(*
Nazwa:			P02_Dispencers
Opis:			Stacja dozownikow
Wersja:			v0.1
Data:			2018-10-10
Autor:			DP
Urzadzenia:		
Konfiguracja:	
Info:

*)
PROGRAM P02_Dispencers
VAR_INPUT
	IbDispencer1DropCatcherBackSensor			AT %I*		:BOOL;					//	Czujnik wycofania tacki kropel dozowników
	IbDispencer2DropCatcherBackSensor 			AT %I*		:BOOL;					//	Czujnik wycofania tacki kropel dozowników
	IbDispencer3DropCatcherBackSensor 			AT %I*		:BOOL;					//	Czujnik wycofania tacki kropel dozowników
	IbDispencer4DropCatcherBackSensor 			AT %I*		:BOOL;					//	Czujnik wycofania tacki kropel dozowników
	IbDispencersCatch1SensorValue 				AT %I*		:DINT;					//	Wejscie czujnika otwarcia siłownika chwytania
	IbDispencersCatch2SensorValue				AT %I*		:DINT;					//	Wejscie czujnika otwarcia siłownika chwytania
	IbDispencersCatch3SensorValue				AT %I*		:DINT;					//	Wejscie czujnika otwarcia siłownika chwytania
	IbDispencersCatch4SensorValue				AT %I*		:DINT;					//	Wejscie czujnika otwarcia siłownika chwytania
	IbDispencersDragLeftLeadBefore1UpSensor		AT %I*		:BOOL;					//	Czujnik
	IbDispencersDragLeftLeadAfter1UpSensor		AT %I*		:BOOL;					//	Czujnik
	IbDispencersDragRightLeadBefore1UpSensor	AT %I*		:BOOL;					//	Czujnik
	IbDispencersDragRightLeadAfter1UpSensor		AT %I*		:BOOL;					//	Czujnik
	IbDispencersDragLeftDragUpSensor 			AT %I*		:BOOL;					// 	Czujnik
	IbDispencersDragLeftDragDownSensor 			AT %I*		:BOOL;					// 	Czujnik
	IbDispencersDragRightDragUpSensor 			AT %I*		:BOOL;					// 	Czujnik
	IbDispencersDragRightDragDownSensor 		AT %I*		:BOOL;					// 	Czujnik
	IbDispencersDragLeftDragHomingSensor 		AT %I*		:BOOL;					//	Czujnik bazowania
	IbDispencersDragRightDragHomingSensor 		AT %I*	 	:BOOL;					//	Czujnik bazowania
	IbDispencerAfterCheckFormSensor				AT %I*		:BOOL; 					//	Czujnik po przecionganiu formatek na ukos
	IbDispencer12NoColisionWhenDosingSensor		AT %I*		:BOOL:=TRUE;			//	Czujnik indukcyjny
	IbDispencer34NoColisionWhenDosingSensor		AT %I*		:BOOL:=TRUE;			//	Czujnik indukcyjny
	//EX
	IbTankLevelHighEX									AT %I*:BOOL;
	IbTankLevelLowEX                                    AT %I*:BOOL;
	IbTankLevelExError									AT %I*:BOOL;
END_VAR
VAR
	
	(*******DOZOWNIK 1*********)
	fbDispencer1										: FB_ServoDispencerServoLifter;			//Blok sterujacy dozownikiem nr1
	eDispencer1State									: E_Station; 							// Stan pracy podajnika platynek			
	eDispencer1RunningState								: E_DispencerState; 
	fbDispencer1State									: FB_State;	
	
	tonDispencer1SuckingValveOpenedSensor				: TON;			//Symulacja czujników 
	tonDispencer1DosingValveOpenedSensor				: TON;			//Symulacja czujników 
	tonDispencer1DosingValveClosedSensor				: TON;			//Symulacja czujników 
	tonDispencer1SuckingValveClosedSensor				: TON;
	
	//WEJŚCIA WYJŚCIA SPRZĘTOWE
	//IbDispencer1SuckingValveOpenedSensor AT%I*:BOOL;	(*dok IO-L*)	//Czujnik otwarcia zaworu ssącego dozownika 1
	QbDispencer1DropCatcherValveActuator				:BOOL;			(*Pneu*)		//Otwarcie tacki
	//IbDispencer1SuckingValveClosedSensor AT%I*:BOOL;	(*dok IO-L*)	//Czujnik zamknięcia zaworu ssąceg odozownika 1
	QbDispencer1SuckingValveActuator					:BOOL;				(*Pneu*)		//sterowanie zaworem ssącego (podłaczenie do wyspypneu)
	QbDispencer1DosingValveActuator						:BOOL;				(*Pneu*)		//sterowanie zaworem dozującym (podłaczenie do wyspypneu)
	
	(*******DOZOWNIK 2*********)
	fbDispencer2										: FB_ServoDispencerServoLifter;				//Blok sterujacy dozownikiem nr 1
	eDispencer2State									: E_Station; 							// Stan pracy podajnika platynek			
	eDispencer2RunningState								: E_DispencerState; 
	fbDispencer2State									: FB_State;	
	
	tonDispencer2SuckingValveOpenedSensor				: TON;			//Symulacja czujników 
	tonDispencer2DosingValveOpenedSensor				: TON;			//Symulacja czujników 
	tonDispencer2DosingValveClosedSensor				: TON;			//Symulacja czujników 
	tonDispencer2SuckingValveClosedSensor				: TON;
	
	//WEJŚCIA WYJŚCIA SPRZĘTOWE
	QbDispencer2DropCatcherValveActuator				:BOOL;			(*Pneu*)			//sterowanie tacką kropel(podłaczenie do wyspy pneu)
	//IbDispencer2SuckingValveOpenedSensor AT%I*:BOOL;	(*dok IO-L*)		//Czujnik otwarcia zaworu ssącego dozownika 1
	//IbDispencer2SuckingValveClosedSensor AT%I*:BOOL;	(*dok IO-L*)		//Czujnik zamknięcia zaworu ssącego dozownika 1
	QbDispencer2SuckingValveActuator					:BOOL;				(*Pneu*)			//sterowanie zaworem ssącego(podłaczeniedowyspypneu)
	QbDispencer2DosingValveActuator						:BOOL;				(*Pneu*)			//sterowanie zaworemd ozującym(podłaczeniedowyspypneu)
	QbDispencerDropCatcherSuck							:BOOL;				(*Pneu*)				//Zasysanie płynu z tacek

	(*******DOZOWNIK 3*********)
	fbDispencer3										: FB_ServoDispencerServoLifter;				//Blok sterujacy dozownikiem nr 1
	eDispencer3State									: E_Station; 							// Stan pracy podajnika platynek			
	eDispencer3RunningState								: E_DispencerState; 
	fbDispencer3State									: FB_State;	
	
	tonDispencer3SuckingValveOpenedSensor				: TON;			//Symulacja czujników 
	tonDispencer3DosingValveOpenedSensor				: TON;			//Symulacja czujników 
	tonDispencer3DosingValveClosedSensor				: TON;			//Symulacja czujników 
	tonDispencer3SuckingValveClosedSensor				: TON;
	
	//WEJŚCIA WYJŚCIA SPRZĘTOWE
	QbDispencer3DropCatcherValveActuator				:BOOL;			(*Pneu*)			//Sterowanie tacką kropel(podłaczenie do wyspy pneu)
	//IbDispencer2SuckingValveOpenedSensor AT%I*:BOOL;	(*dok IO-L*)		//Czujnik otwarcia zaworu ssącego dozownika 1
	//IbDispencer2SuckingValveClosedSensor AT%I*:BOOL;	(*dok IO-L*)		//Czujnik zamknięcia zaworu ssącego dozownika 1
	QbDispencer3SuckingValveActuator					:BOOL;				(*Pneu*)			//sterowanie zaworem ssącego(podłaczeniedowyspypneu)
	QbDispencer3DosingValveActuator						:BOOL;				(*Pneu*)			//sterowanie zaworemd ozującym(podłaczeniedowyspypneu)

	(*******DOZOWNIK 4*********)
	fbDispencer4										: FB_ServoDispencerServoLifter;			// Blok sterujacy dozownikiem nr 1
	eDispencer4State									: E_Station; 							// Stan pracy podajnika platynek			
	eDispencer4RunningState								: E_DispencerState; 
	fbDispencer4State									: FB_State;	
	
	tonDispencer4SuckingValveOpenedSensor				: TON;			//Symulacja czujników 
	tonDispencer4DosingValveOpenedSensor				: TON;			//Symulacja czujników 
	tonDispencer4DosingValveClosedSensor				: TON;			//Symulacja czujników 
	tonDispencer4SuckingValveClosedSensor				: TON;
	
	//WEJŚCIA WYJŚCIA SPRZĘTOWE
	QbDispencer4DropCatcherValveActuator				:BOOL;			(*Pneu*)			//sterowanie tacką kropel(podłaczenie do wyspy pneu)
	//IbDispencer2SuckingValveOpenedSensor AT%I*:BOOL;	(*dok IO-L*)		//Czujnik otwarcia zaworu ssącego dozownika 1
	//IbDispencer2SuckingValveClosedSensor AT%I*:BOOL;	(*dok IO-L*)		//Czujnik zamknięcia zaworu ssącego dozownika 1
	QbDispencer4SuckingValveActuator					:BOOL;				(*Pneu*)			//sterowanie zaworem ssącego(podłaczeniedowyspypneu)
	QbDispencer4DosingValveActuator						:BOOL;				(*Pneu*)			//sterowanie zaworemd ozującym(podłaczeniedowyspypneu)
	
	(*******PODNOSNIK TACKI I CHWYTAKA*********)
	fbDispencersCatch1Station							:FB_CatchStationWithSensor;			// Blok stacji chwytaka dozowników
	fbDispencersCatch2Station							:FB_CatchStationWithSensor;			// Blok stacji chwytaka dozowników
	fbDispencersCatch3Station							:FB_CatchStationWithSensor;			// Blok stacji chwytaka dozowników
	fbDispencersCatch4Station							:FB_CatchStationWithSensor;			// Blok stacji chwytaka dozowników
	eDispencersCatch1State								:E_Station; 				// Stan chwytaka stabilizujšcego pod podajnikiem platynek
	eDispencersCatch2State								:E_Station; 				// Stan chwytaka stabilizujšcego pod podajnikiem platynek
	eDispencersCatch3State								:E_Station; 				// Stan chwytaka stabilizujšcego pod podajnikiem platynek
	eDispencersCatch4State								:E_Station; 				// Stan chwytaka stabilizujšcego pod podajnikiem platynek
	eDispencersCatch1RunningState						:E_CatchStationState; 		// Poprzedni stan chwytaka pod podajnikiem nakrętek
	eDispencersCatch2RunningState						:E_CatchStationState; 		// Poprzedni stan chwytaka pod podajnikiem nakrętek
	eDispencersCatch3RunningState						:E_CatchStationState; 		// Poprzedni stan chwytaka pod podajnikiem nakrętek
	eDispencersCatch4RunningState						:E_CatchStationState; 		// Poprzedni stan chwytaka pod podajnikiem nakrętek
	fbDispencersCatch1State								:FB_State;
	fbDispencersCatch2State								:FB_State;
	fbDispencersCatch3State								:FB_State;
	fbDispencersCatch4State								:FB_State;
	
//WEJSCIA I WYJSCIA SPRZETOWE
	QbDispencersCatch1HeightUpCmd 				AT %Q*	:BOOL; 			(*PLC.A17*)		// Wyjście sterujące podnośnikiem chwytaka i tacki dozownika , Silnik w górę
	QbDispencersCatch1HeightDownCmd 			AT %Q*	:BOOL; 		(*PLC.A17*)		// Wyjście sterujące podnośnikiem chwytaka i tacki dozownika, Silnik w dół
	IbDispencersCatch1HeightEncoderPulses 		AT %I*	:BOOL;	(*PLC.A13*)
	
	IbDispencersCatchHeightEncoderSetCDone		AT %I*: BOOL;
	IudiDispencersCatchHeightEncoderCV          AT %I*: UDINT; 
	QbDispencersCatchHeightEncoderSetC 			AT %Q*: BOOL;		
	QudiDispencersCatchHeightEncoderSetCV       AT %Q*: UDINT; 	
	                                            	
	                                            	
	
	
	QbDispencersCatch1Actuator 							:BOOL;					(*Pneu*)		// Wyjście sterujące chwytakiem pod dozownikami
	QbDispencersCatch2Actuator 							:BOOL;					(*Pneu*)		// Wyjście sterujące chwytakiem pod dozownikami
	QbDispencersCatch3Actuator 							:BOOL;					(*Pneu*)		// Wyjście sterujące chwytakiem pod dozownikami
	QbDispencersCatch4Actuator 							:BOOL;					(*Pneu*)		// Wyjście sterujące chwytakiem pod dozownikami

	QbDispencersCatchMaxPressure						:BOOL;				(*Pneu*)			//sterowanie zaworemd ozującym(podłaczeniedowyspypneu)
	
	(*****************SZLABANY*******************)
	fbDispencerGatesStation								:FB_EntranceGatesServo;			// Blok stacji szlabanów 
		
	(*******PRZECIAGANIE**********)
	eDispencersDragLeftStation							: E_Station;
	eDispencersDragLeftRunningStation					: E_DragStationState;
	fbDispencersDragLeftState							: FB_State;
	eDispencersDragRightStation							: E_Station;
	eDispencersDragRightRunningStation					: E_DragStationState;
	fbDispencersDragRightState							: FB_State;	
	fbDispencersDragLeftStation							: FB_FormsDragStepper;	
	fbDispencersDragRightStation						: FB_FormsDragStepper;
	
	//WEJSCIA I WYJSCIA SPRZETOWE
	
	QbDispencersDragLeftDragActuator                   :BOOL;						// Siłownikiem przeciągania (1 faza)
	
	QbDispencersDragLeftLeadBefore1Actuator          :BOOL;							// Siłownikiem prowadzenia przed 1(1 faza)
	QbDispencersDragLeftLeadAfter1Actuator          :BOOL;							// Siłownikiem prowadzenia przed 1(1 faza)
	
	QbDispencersDragRightDragActuator                  :BOOL;						// Siłownikiem przeciągania (1 faza)
	
	QbDispencersDragRightLeadBefore1Actuator          :BOOL;						// Siłownikiem prowadzenia przed 2(1 faza)	
	QbDispencersDragRightLeadAfter1Actuator          :BOOL;							// Siłownikiem prowadzenia przed 1(1 faza)
		
	(**********ZBIORNIKI**************)
	//Zbiornik
	IbTank1LevelLow 							 AT %I* :BOOL; 				(*PLC.A8*)	// Niski poziom masy w zbiorniku
	IbTank2LevelLow 							 AT %I* :BOOL; 				(*PLC.A8*)	// Niski poziom masy w zbiorniku
	QbTank1LevelSensorCalibration 			     AT %Q* :BOOL;  (*PLC.A20*)	// Kalibracja czujnika poziomu leja nr 1
	QbTank2LevelSensorCalibration 				 AT %Q* :BOOL;  (*PLC.A20*)	// Kalibracja czujnika poziomu leja nr 2
	
	
	QbTank1Pressure								 AT %Q* :BOOL;						(*Pneu*)	// Ciśnienie w zbiorniku nr 1
	bTank1LevelLow                                      :BOOL;									// Sygnały sterujące pompy 1 zależnie od ich odwrócenia
	bTank2LevelLow										:BOOL;									// Sygnały sterujące pompy 2 zależnie od ich odwrócenia
	
	//Pompa podająca
	QbTank1PumpStart 							AT %Q*	:BOOL;		(*PLC.A21*)	//Załączenie pompy masy do zbiornika
	QbTank2PumpStart 							AT %Q*	:BOOL;		(*PLC.A21*)	//Załączenie pompy masy do zbiornika
	QbTank3PumpStart 							AT %Q*	:BOOL;		(*PLC.A21*)	//Załączenie pompy masy do zbiornika
	QbTank4PumpStart 							AT %Q*	:BOOL;		(*PLC.A21*)	//Załączenie pompy masy do zbiornika
	IbTank1PumpFuseOK 							AT %I*  :BOOL; 				//Potwierdzenie z zabezpieczenia pompy 1 - OK
	IbTank2PumpFuseOK 							AT %I*  :BOOL; 				//Potwierdzenie z zabezpieczenia pompy 2 - OK
	IbTank3PumpFuseOK 							AT %I*  :BOOL; 				//Potwierdzenie z zabezpieczenia pompy 2 - OK
	IbTank4PumpFuseOK 							AT %I*  :BOOL; 				//Potwierdzenie z zabezpieczenia pompy 2 - OK
		
	(*GRZAŁKA ZBIORNIKA*)
	fbTankHeating										: FB_TankHeating;	
	eTankHeatingState									: E_Station; 					// Stan pracy grzania
	eTankHeatingRunningState							: E_MassHeatingState; 			// Stan pracy grzania
	fbTankHeatingState									: FB_State;
		
	//WEJŚĆIA I WYJŚĆIA SPRZĘTOWE		
	QbTankHeatingPWMOut							AT %Q* :BOOL; 					// Wyjście sterujące temperaturą grzałki
	AInTankHeatingTempCVSensor 					AT %I* :INT; 			// Wartość aktualnej temperatury grzałki
	IbTankHeatingTempSensorFailure 				AT %I* :BOOL;  		// Informacja o uszkodzeniu czujnika temperatury grzałki	
	
	//Mieszadło zbiornika
	IbFuseTankMixerEngineOK						AT %I* :BOOL;	(*PLC.A7*)	//Bezpiecznik silnika mieszadła OK
	IbFuseTankMixerEngineWorking				AT %I* :BOOL;	{warning 'oprogramowac nowy sygnał mieszadla'}			//Potwierdzenie pracy silnika mieszadła OK	
	QbTank1MixerStart 							AT %Q* :BOOL;			(*PLC.A20*)	//Załączenie mieszadła masy do zbiornika
	
	// Zezwolenie na pracę mieszadła zbiornikowego
	tonTank1LevelSensor									: TON;
	
	tofTank2LevelSensor									: TOF;
	tonTank2LevelSensor									: TON;
	
	tonTank1LevelWarning	   							: TON;
	tonTank2LevelWarning	   							: TON;
	
	tonTank1EmptyAlarm									: TON;
	tonTank2EmptyAlarm									: TON;
	rtDispencer1DoseDone								: R_TRIG;
	rtDispencer2DoseDone								: R_TRIG;
	
	tonTankLevelSensorCalibrationLight					: TON;
	tonTankLevelSensorCalibrationDark					: TON;
	
	(**********OSLONA DOZOWNIKOW*************)	
	
	nCalibrationDialog								 	: INT;

	TimerDispencer1Enable								: TOF;
	TimerDispencer2Enable								: TOF;
	TimerDispencer3Enable								: TOF;
	TimerDispencer4Enable								: TOF;		
	
	(*Wykres dozowania*)
	fbDosingChart1										: FB_WriteDataToArrayString;
	fbDosingChart2										: FB_WriteDataToArrayString;
	fbDosingChart3										: FB_WriteDataToArrayString;
	fbDosingChart4										: FB_WriteDataToArrayString;
	fbDosingStChart1									: FB_WriteDataToArrayOfArrays;
	fbDosingStChart2									: FB_WriteDataToArrayOfArrays;
	fbDosingStChart3									: FB_WriteDataToArrayOfArrays;
	fbDosingStChart4									: FB_WriteDataToArrayOfArrays;
	nChartCycleTime										: INT;
	tDelayDispencerValve								: TIME;

	rtEnable											: R_TRIG;

	fbDropCatcherSuck									: FB_Blink_AS;
	nDose1Counter										: INT;
	nDose2Counter										: INT;
	nDose1CounterWhenLowLevel							: INT;
	nDose2CounterWhenLowLevel							: INT;	
	nDoseCounter1										: INT;
	nDoseCounter2										: INT;	
	// Czujnik poziomu masy przewodząco pojmenościowy LiquiPoint FTW33
	// Zmienne akcji ACT_ConductiveMassSensor
	
	bTank1LevelLowConductiveSensor						: BOOL;
	bTank1SensorDiagnosis								: BOOL;     // Diagnostyka czujnika
	IusiTank1SensorValue0						AT%I*	: USINT;
	IusiTank1SensorValue1						AT%I*	: USINT;
	IusiTank1SensorValue2						AT%I*	: USINT;
	IusiTank1SensorValue3						AT%I*	: USINT;
	IusiTank1SensorDiagnosis					AT%I*	: USINT;
    iTank1Sensor1Value									: INT;	                         
	tonTank1LevelLowConductiveSensor					: TON;
	iTank1Sensor1ValueTemp								: INT;	
	
	bTank2LevelLowConductiveSensor						: BOOL;
	bTank2SensorDiagnosis								: BOOL;     // Diagnostyka czujnika
	IusiTank2SensorValue0						AT%I*	: USINT;
	IusiTank2SensorValue1						AT%I*	: USINT;
	IusiTank2SensorValue2						AT%I*	: USINT;
	IusiTank2SensorValue3						AT%I*	: USINT;
	IusiTank2SensorDiagnosis					AT%I*	: USINT;    
	iTank2Sensor1Value									: INT;		                              
	tonTank2LevelLowConductiveSensor					: TON;	
	iTank2Sensor1ValueTemp								: INT;
	
	//Filtrowanie sygnału
	fbFilterExiTank1Sensor1Value						: FB_FilterEx;
	
	tonMixerNotWorking									: TON;
	
	tonTank1PumpFuseOK									: TON;
	tonTank2PumpFuseOK									: TON;
	
	// Pomocnicze do hamulców
	bDispencer1ManualBrakeOff							: BOOL;
	bDispencer2ManualBrakeOff							: BOOL;	
	bDispencer3ManualBrakeOff							: BOOL;
	bDispencer4ManualBrakeOff							: BOOL;
	
	aDispenser1VirtualLifter							: AXIS_REF;
	aDispenser2VirtualLifter							: AXIS_REF;
	aDispenser3VirtualLifter							: AXIS_REF;
	aDispenser4VirtualLifter							: AXIS_REF;
	
	bDispencer1WithLifter								: BOOL;
	bDispencer2WithLifter								: BOOL;
	bDispencer3WithLifter								: BOOL;
	bDispencer4WithLifter								: BOOL;
	bDispenser1LifterMaster								: BOOL;
	bDispenser2LifterMaster								: BOOL;
	bDispenser3LifterMaster								: BOOL;
	bDispenser4LifterMaster								: BOOL;	
	
	bDispencer12MultiMasterSync							: BOOL;  //Do synchronizacji dozownikow 1-2 miedzy sobą
	bDispencer34MultiMasterSync							: BOOL;	//Do synchornizacji dozownikow 3-4 między sobą
	//bDispencersSyncSim									:BOOL;
	bDispenser1MultiMasterSyncOut						: BOOL;	// Wyjscie synchronizacji dozownika z pozostałymi dozownikami na podnośniku
	bDispenser2MultiMasterSyncOut						: BOOL;	// Wyjscie synchronizacji dozownika z pozostałymi dozownikami na podnośniku
	bDispenser3MultiMasterSyncOut						: BOOL;	// Wyjscie synchronizacji dozownika z pozostałymi dozownikami na podnośniku
	bDispenser4MultiMasterSyncOut						: BOOL;	// Wyjscie synchronizacji dozownika z pozostałymi dozownikami na podnośniku
	
	bDispencer1Manual									: BOOL;
	bDispencer2Manual									: BOOL;
	bDispencer3Manual									: BOOL;
	bDispencer4Manual									: BOOL;
	
	bDispencer1DropCatcherValveActuator					: BOOL;
	bDispencer2DropCatcherValveActuator					: BOOL;
	bDispencer3DropCatcherValveActuator					: BOOL;
	bDispencer4DropCatcherValveActuator					: BOOL;
	
	ftChangeover										: F_TRIG;
	
	//Mikołaj
	
	rtbDispencer12EnableShow							: R_TRIG;
	ftbDispencer12EnableShow							: F_TRIG;
	rtbDispencer34EnableShow							: R_TRIG;
	ftbDispencer34EnableShow							: F_TRIG;
	
	fbDispencersCleaningPID								: FB_PIDBasic;
	tonbDispencer12Cleaning								: TON;
	tonbDispencer34Cleaning								: TON;	
	fbDispencersCIP										: FB_InputFilter;

	ftCIP												: F_TRIG;
	tonbCIP												: TON;
	ftbCIP												: F_TRIG;
	rtbCIP												: R_TRIG;
	
	tonResetOpenCalibration								: TON;
	tonResetCloseCalibration							: TON;
	
	tofDispencersDragLeftStationEnable					: TOF;
	tofDispencersDragRightStationEnable					: TOF;	
	
	
	fbFormsDragingStepperState: INT;
	eState: INT;

	tofTank1LevelSensor: TOF;
//dodane filtry 	
	fbIbDispencer1DropCatcherBackSensor	:FB_InputFilter;
	fbIbDispencer2DropCatcherBackSensor	:FB_InputFilter;
	fbIbDispencer3DropCatcherBackSensor	:FB_InputFilter;
	fbIbDispencer4DropCatcherBackSensor	:FB_InputFilter;
		
	arTemp:AXIS_REF;

	(*Tryb serwisowy dozownikow*)
	ftbDispencersPullingSlow: F_TRIG;
	ftbDispencersPullingFast: F_TRIG;
	ftbDispencersPullingSlowContinous: F_TRIG;
	ftbDispencersPullingFastContinous: F_TRIG;	
	ftbDispencersLifterUp: F_TRIG;
	ftbDispencersLifterDown: F_TRIG;
	tonbDispencersPullingContinous: TON;

	rtDispencer1Sync												: R_TRIG;
	rtDispencer2Sync												: R_TRIG;
	rtDispencer3Sync												: R_TRIG;
	rtDispencer4Sync												: R_TRIG;
	fbDispencer1Sync												: FB_InputFilter_v2;	
	fbDispencer2Sync												: FB_InputFilter_v2;	
	fbDispencer3Sync												: FB_InputFilter_v2;	
	fbDispencer4Sync												: FB_InputFilter_v2;	
	tofDispencersSync												: TOF;
	rtManualMode													: R_TRIG;
	ftManualMode													: F_TRIG;
	rtbDispencer1Sync												: R_TRIG;	
	rtbDispencer2Sync												: R_TRIG;		
	rtbDispencer3Sync												: R_TRIG;	
	rtbDispencer4Sync												: R_TRIG;	
	rtbDispencer12Sync												: R_TRIG;
	rtbDispencer34Sync												: R_TRIG;
	rtbDispencer1234Sync											: R_TRIG;	
	rtHeightSetDispencer12											: R_TRIG;
	rtHeightSetDispencer34											: R_TRIG;

	bDispencer1SyncTemp												: BOOL;
	bDispencer2SyncTemp												: BOOL;
	bDispencer3SyncTemp												: BOOL;
	bDispencer4SyncTemp												: BOOL;
	
	(*Reset warningów*)
	tonDispencersWarningReset : TON;
	
	(*Podtrzymanie receptur*)
	bFormsDragingLeftEnableDelay: BOOL;
	bFormsDragingRightEnableDelay: BOOL;
	bDispencer1EnableDelay: BOOL;
	bDispencer2EnableDelay: BOOL;
	bDispencer3EnableDelay: BOOL;
	bDispencer4EnableDelay: BOOL;
	
	(*inne*)
	btemp					:BOOL;
	
	(*Ex*)
	tonLowLevelExSensor		:TON;
	tonErrorExSensorDelay	:TON;
	bTank1LevelExSensor: BOOL;	

	//Zmienne od EVENTLOGGER
	bAlarmInit 						: BOOL := TRUE; 
	nAlarmNumerator					: INT;
	arfbAlarm						: ARRAY[0..19] OF  FB_TcAlarm;		//Tablica bloczków błędów
	fbSourceInfo 					: FB_TcSourceInfo;
	iSourceInfo						: I_TcSourceInfo;
	sAlarmTest						: STRING;
	//Koniec zmiennych od EVENTLOGGER
END_VAR

(* Temp zbiornika*)
VIS.lrTankHeatingTempCV := AInTankHeatingTempCVSensor/10.0;
(* Koniec Temp zbiornika*)

fbIbDispencer1DropCatcherBackSensor(bIN:=IbDispencer1DropCatcherBackSensor AND IbDispencer2DropCatcherBackSensor ,tFilterTimeOn:=T#20MS,tFilterTimeOff:=T#20MS,bOUT=>);
fbIbDispencer2DropCatcherBackSensor(bIN:=IbDispencer2DropCatcherBackSensor AND IbDispencer1DropCatcherBackSensor,tFilterTimeOn:=T#20MS,tFilterTimeOff:=T#20MS,bOUT=>);
fbIbDispencer3DropCatcherBackSensor(bIN:=IbDispencer3DropCatcherBackSensor AND IbDispencer4DropCatcherBackSensor,tFilterTimeOn:=T#20MS,tFilterTimeOff:=T#20MS,bOUT=>);
fbIbDispencer4DropCatcherBackSensor(bIN:=IbDispencer4DropCatcherBackSensor AND IbDispencer3DropCatcherBackSensor,tFilterTimeOn:=T#20MS,tFilterTimeOff:=T#20MS,bOUT=>);
	


(***Skalownaie wartości zadanej na 1-100%************)
(*
:=DINT_TO_USINT(
	F_Scaling(
	rValue:= LREAL_TO_DINT(lrFormsDragingLeftVelocity), 
	rXmin:= 1, 
	rXmax:= 1000, 
	rYmin:= 1, 
	rYmax:= 10)
	)
;*)


fbDispencersCatch1Station.lrSensorTolerance:= fbDispencersCatch2Station.lrSensorTolerance:= 
fbDispencersCatch3Station.lrSensorTolerance:= fbDispencersCatch4Station.lrSensorTolerance:= 
	F_Scaling(
	rValue:= LREAL_TO_DINT(lrDispencersCatchTolerance*10), 
	rXmin:= 1, 
	rXmax:= 100, 
	rYmin:= 100, 
	rYmax:= 10000)
;

IF lrDispencersCatchTolerance = 100 THEN
	fbDispencersCatch1Station.lrSensorTolerance	:= fbDispencersCatch2Station.lrSensorTolerance	:= 100000;	
	fbDispencersCatch3Station.lrSensorTolerance	:= fbDispencersCatch4Station.lrSensorTolerance	:= 100000;	
END_IF
(****Koniec skalownaie wartości zadanej na 1-100%****)

//Grzanie zbiornika
IF NOT VIS.bLidFeederEnableShow THEN
	//GVL.bDispencersCatchEnable																		:= NOT VIS.bSimulation ;
END_IF
(**SYMULACJA CZUJNIKÓW IGLIC**)
tDelayDispencerValve																			:= T#50MS;

tonDispencer1SuckingValveClosedSensor(IN:=NOT QbDispencer1SuckingValveActuator, PT:=tDelayDispencerValve);
tonDispencer1SuckingValveOpenedSensor(IN:=QbDispencer1SuckingValveActuator,PT:=tDelayDispencerValve);
tonDispencer1DosingValveOpenedSensor(IN:=QbDispencer1DosingValveActuator ,PT:=tDelayDispencerValve);
tonDispencer1DosingValveClosedSensor(IN:=NOT QbDispencer1DosingValveActuator ,PT:=tDelayDispencerValve);

tonDispencer2SuckingValveClosedSensor(IN:=NOT QbDispencer2SuckingValveActuator, PT:=tDelayDispencerValve);
tonDispencer2SuckingValveOpenedSensor(IN:=QbDispencer2SuckingValveActuator,PT:=tDelayDispencerValve);
tonDispencer2DosingValveOpenedSensor(IN:=QbDispencer2DosingValveActuator ,PT:=tDelayDispencerValve);
tonDispencer2DosingValveClosedSensor(IN:=NOT QbDispencer2DosingValveActuator ,PT:=tDelayDispencerValve);

tonDispencer3SuckingValveClosedSensor(IN:=NOT QbDispencer3SuckingValveActuator, PT:=tDelayDispencerValve);
tonDispencer3SuckingValveOpenedSensor(IN:=QbDispencer3SuckingValveActuator,PT:=tDelayDispencerValve);
tonDispencer3DosingValveOpenedSensor(IN:=QbDispencer3DosingValveActuator ,PT:=tDelayDispencerValve);
tonDispencer3DosingValveClosedSensor(IN:=NOT QbDispencer3DosingValveActuator ,PT:=tDelayDispencerValve);

tonDispencer4SuckingValveClosedSensor(IN:=NOT QbDispencer4SuckingValveActuator, PT:=tDelayDispencerValve);
tonDispencer4SuckingValveOpenedSensor(IN:=QbDispencer4SuckingValveActuator,PT:=tDelayDispencerValve);
tonDispencer4DosingValveOpenedSensor(IN:=QbDispencer4DosingValveActuator ,PT:=tDelayDispencerValve);
tonDispencer4DosingValveClosedSensor(IN:=NOT QbDispencer4DosingValveActuator ,PT:=tDelayDispencerValve);
(**Koniec SYMULACJA CZUJNIKÓW IGLIC*)

aLimits();
aAntyColision();
aDispencersEnable();
aCleaning();
aDispencersLiftersBefore(); //musi być odpowednia kolejność 
aDispencersManualMode();
aDispencer1();
aDispencer2();
aDispencer3();
aDispencer4();
aDispencersLiftersAfter();
aDispencerCatch1();
aDispencerCatch2();
aDispencerCatch3();
aDispencerCatch4();
aDispencerCatchPressure();
aDispencersCatchWarnings();
aDropCatcher();
aDispencerDragStation();
aDispencersDragStationLeadActuators();
aTanks();
aTanksRainbowMode();
aTankWarning();
aTankHeating();
aTDRMassSensor();
aExSensor();
aLevelSensorCalibration();
aDosingChartHMI(); //Przygotowanie danych do wykresu

(* BAZOWANIE - ZMIAN*)
rtEnable		(CLK:=fbDispencer1.bEnable OR fbDispencer2.bEnable OR fbDispencer3.bEnable OR fbDispencer4.bEnable,				Q=>);
ftChangeover	(CLK:=fbDispencer1.bChangeover OR fbDispencer2.bChangeover OR fbDispencer2.bChangeover OR fbDispencer2.bChangeover, Q=>);
ftCIP			(CLK:=bCIP, 																									Q=>);

IF ( rtEnable.Q  OR ftChangeover.Q OR ftCIP.Q) AND (P00_PackML.fbPMLAuto.ePMLState = E_PMLState.ePMLState_IDLE OR P00_PackML.fbPMLAuto.ePMLState = E_PMLState.ePMLState_EXECUTE)  THEN
	VIS.bDispencer12LifterHeightSet:=TRUE;
	VIS.bDispencer34LifterHeightSet:=TRUE;	
	VIS.bDispencersCatchHeightSet:=TRUE;
	
ELSIF ( fbDispencer1.eState=E_Station.eHomingDone AND 
		fbDispencer2.eState=E_Station.eHomingDone AND 
		fbDispencer3.eState=E_Station.eHomingDone AND 
		fbDispencer4.eState=E_Station.eHomingDone) OR 
		VIS.bErrorOccure THEN
	VIS.bDispencer12LifterHeightSet:=FALSE;
	VIS.bDispencer34LifterHeightSet:=FALSE;
ELSIF fbDispencersCatch1Station.eState=E_Station.eHomingDone OR VIS.bErrorOccure THEN
	VIS.bDispencersCatchHeightSet:=FALSE;
ELSIF fbDispencer1.eState=E_Station.eHomingDone OR VIS.bErrorOccure THEN
	VIS.bDispencer12LifterHeightSet:=FALSE;
ELSIF fbDispencer2.eState=E_Station.eHomingDone OR VIS.bErrorOccure THEN
	VIS.bDispencer12LifterHeightSet:=FALSE;
ELSIF fbDispencer3.eState=E_Station.eHomingDone OR VIS.bErrorOccure THEN
	VIS.bDispencer34LifterHeightSet:=FALSE;
ELSIF fbDispencer4.eState=E_Station.eHomingDone OR VIS.bErrorOccure THEN
	VIS.bDispencer34LifterHeightSet:=FALSE;

END_IF


(********* GENEROWANIE STANU STACJI DO WIZKI**********)
fbDispencersDragLeftState(
	eState:=eDispencersDragLeftStation, 
	bRun:=VIS.bFormsDragingLeftRun,
	eFormsDragingRunningState:=eDispencersDragLeftRunningStation , 
	sStateDesc=> VIS.sFormsDragingLeftState,
	iState=>VIS.iFormsDragingLeftState);
fbDispencersDragRightState(
	eState:=eDispencersDragRightStation, 
	bRun:=VIS.bFormsDragingRightRun,
	eFormsDragingRunningState:=eDispencersDragRightRunningStation , 
	sStateDesc=> VIS.sFormsDragingRightState,
	iState=>VIS.iFormsDragingRightState);	
fbDispencer1State(
	eState:=eDispencer1State , 
	bRun:=VIS.bDispencer1Dose,
	eDispencerRunningState:=eDispencer1RunningState , 
	sStateDesc=> VIS.sDispencer1State,
	iState=>VIS.iDispencer1State);
fbDispencer2State(
	eState:=eDispencer2State , 
	bRun:=VIS.bDispencer2Dose,
	eDispencerRunningState:=eDispencer2RunningState , 
	sStateDesc=> VIS.sDispencer2State,
	iState=>VIS.iDispencer2State);
fbDispencer3State(
	eState:=eDispencer3State , 
	bRun:=VIS.bDispencer3Dose,
	eDispencerRunningState:=eDispencer3RunningState , 
	sStateDesc=> VIS.sDispencer3State,
	iState=>VIS.iDispencer3State);
fbDispencer4State(
	eState:=eDispencer4State , 
	bRun:=VIS.bDispencer4Dose,
	eDispencerRunningState:=eDispencer4RunningState , 
	sStateDesc=> VIS.sDispencer4State,
	iState=>VIS.iDispencer4State);
fbDispencersCatch1State(
	eState:=eDispencersCatch1State	 , 
	bRun:=VIS.bDispencers1Catch,	
	eCatchRunningState:=eDispencersCatch1RunningState , 
	sStateDesc=> VIS.sDispencersCatch1State,
	iState=>VIS.iDispencersCatch1State	);		
fbDispencersCatch2State(
	eState:=eDispencersCatch2State	 , 
	bRun:=VIS.bDispencers2Catch,	
	eCatchRunningState:=eDispencersCatch2RunningState , 
	sStateDesc=> VIS.sDispencersCatch2State,
	iState=>VIS.iDispencersCatch2State	);	
fbDispencersCatch3State(
	eState:=eDispencersCatch3State	 , 
	bRun:=VIS.bDispencers3Catch,	
	eCatchRunningState:=eDispencersCatch3RunningState , 
	sStateDesc=> VIS.sDispencersCatch3State,
	iState=>VIS.iDispencersCatch3State	);	
fbDispencersCatch4State(
	eState:=eDispencersCatch4State	 , 
	bRun:=VIS.bDispencers4Catch,	
	eCatchRunningState:=eDispencersCatch4RunningState , 
	sStateDesc=> VIS.sDispencersCatch4State,
	iState=>VIS.iDispencersCatch4State	);		
fbTankHeatingState(
	eState:=eTankHeatingState, 
	bRun:=bTankHeatingEnable,
	eMassHeatingRunningState:=eTankHeatingRunningState , 
	);
(***** KONIEC GENEROWANIE STANU STACJI DO WIZKI*******)


(**Przypisanie maksymalnej prędkość podnośników dozowników do ekranu ustawiania wykresu dozowania*)
VIS.iHMIDispencersLifterMaxSpeed := 313;
(**Koniec Przypisanie maksymalnej prędkość podnośników dozowników do ekranu ustawiania wykresu dozowania*)


(******* Wypracowanie sygnałów dla HMI *******)
VIS.lrDispencer1ActPos := aDispencer1AxisRef.NcToPlc.ActPos;
VIS.lrDispencer2ActPos := aDispencer2AxisRef.NcToPlc.ActPos;
VIS.lrDispencer3ActPos := aDispencer3AxisRef.NcToPlc.ActPos;
VIS.lrDispencer4ActPos := aDispencer4AxisRef.NcToPlc.ActPos;

(*******Jezeli dwufazowe to przepisuj sygnały**************)


IF NOT VIS.bDosingTwoPhasesShow THEN
	VIS.lrDispencer2DoseVolumeShow:=VIS.lrDispencer1DoseVolumeShow;
	VIS.lrDispencer2Phase1VolumeShow:=VIS.lrDispencer1Phase1VolumeShow;
	VIS.lrDispencer2Phase2VolumeShow:=VIS.lrDispencer1Phase2VolumeShow;
	VIS.lrDispencer2Phase1VelocityShow:=VIS.lrDispencer1Phase1VelocityShow;
	VIS.lrDispencer2Phase2VelocityShow:=VIS.lrDispencer1Phase2VelocityShow;
	VIS.lrDispencer2Phase3VelocityShow:=VIS.lrDispencer1Phase3VelocityShow;
	VIS.lrDispencer2SuckVelocityShow:=VIS.lrDispencer1SuckVelocityShow;
	VIS.lrDispencer2Phase1AccelerationShow:=VIS.lrDispencer1Phase1AccelerationShow;
	VIS.lrDispencer2Phase2AccelerationShow:=VIS.lrDispencer1Phase2AccelerationShow;
	VIS.lrDispencer2Phase3AccelerationShow:=VIS.lrDispencer1Phase3AccelerationShow;
	VIS.lrDispencer2SuckAccelerationShow:=VIS.lrDispencer1SuckAccelerationShow;
	VIS.lrDispencer2Phase1DecelerationShow:=VIS.lrDispencer1Phase1DecelerationShow;
	VIS.lrDispencer2Phase2DecelerationShow:=VIS.lrDispencer1Phase2DecelerationShow;
	VIS.lrDispencer2Phase3DecelerationShow:=VIS.lrDispencer1Phase3DecelerationShow;
	VIS.udiDispencer2DosingDoneDelayTimeShow:=VIS.udiDispencer1DosingDoneDelayTimeShow;
	VIS.lrDispencer2SuckValveOpenVolumeShow:=VIS.lrDispencer1SuckValveOpenVolumeShow;
	VIS.lrDispencer2SuckValveOpenTimeDelayShow:=VIS.lrDispencer1SuckValveOpenTimeDelayShow;
	VIS.lrDispencer2SuckValveCloseVolumeShow:=VIS.lrDispencer1SuckValveCloseVolumeShow;
	VIS.lrDispencer2SuckValveCloseTimeDelayShow:=VIS.lrDispencer1SuckValveCloseTimeDelayShow;
	VIS.lrDispencer2DoseValveOpenVolumeShow:=VIS.lrDispencer1DoseValveOpenVolumeShow;
	VIS.lrDispencer2DoseValveOpenTimeAccShow:=VIS.lrDispencer1DoseValveOpenTimeAccShow;
	VIS.lrDispencer2DoseValveCloseVolumeShow:=VIS.lrDispencer1DoseValveCloseVolumeShow;
	VIS.lrDispencer2DoseValveCloseTimeDecShow:=VIS.lrDispencer1DoseValveCloseTimeDecShow;
	VIS.lrDispencer2DoseSuckingVolumeShow:=VIS.lrDispencer1DoseSuckingVolumeShow;
	VIS.lrDispencer2DoseSuckingTimeDelayShow:=VIS.lrDispencer1DoseSuckingTimeDelayShow;
	VIS.bDispencer2DoseSuckingShow:=VIS.bDispencer1DoseSuckingShow;
	VIS.bDispencer2LiftSynchroPh1Show:=VIS.bDispencer1LiftSynchroPh1Show;
	VIS.bDispencer2LiftSynchroPh2Show:=VIS.bDispencer1LiftSynchroPh2Show;
	VIS.bDispencer2LiftSynchroPh3Show:=VIS.bDispencer1LiftSynchroPh3Show;
	VIS.lrDispencer2LifterStartDosePositionShow:=VIS.lrDispencer1LifterStartDosePositionShow;
	VIS.lrDispencer2LifterStopDosePositionShow:=VIS.lrDispencer1LifterStopDosePositionShow;
	VIS.lrDispencer2LifterVelocityShow:=VIS.lrDispencer1LifterVelocityShow;
	VIS.lrDispencer2LifterAccelerationShow:=VIS.lrDispencer1LifterAccelerationShow;
	VIS.lrDispencer2LifterDecelerationShow:=VIS.lrDispencer1LifterDecelerationShow;
	
//dodane po testach 	
	VIS.lrFormsDragingRightAccelerationShow:=VIS.lrFormsDragingLeftAccelerationShow;
	VIS.lrFormsDragingRightDecelerationShow:=VIS.lrFormsDragingLeftDecelerationShow;
	VIS.lrFormsDragingRightVelocityShow:=VIS.lrFormsDragingLeftVelocityShow;
	
END_IF

IF bCycleReseting THEN
	;
END_IF


(*Opoznienie wyłączanie enabla dozownikow*)
(*Nie zdarzy wyjśc z Disabled podczas zmiany recepptury*)
TimerDispencer1Enable(IN:=bDispencer1Enable OR bDispencer1EnableDelay, PT:=T#5S);
TimerDispencer2Enable(IN:=bDispencer2Enable OR bDispencer2EnableDelay, PT:=T#5S);
TimerDispencer3Enable(IN:=bDispencer3Enable OR bDispencer3EnableDelay, PT:=T#5S);
TimerDispencer4Enable(IN:=bDispencer4Enable OR bDispencer4EnableDelay, PT:=T#5S);
// Dodatkowe podtrzymanie przy zmianie receptury
IF  P00_PackML.fbbRecipeLoading.bOut AND GVL.bDispencer1Enable	THEN	bDispencer1EnableDelay	:= 	TRUE;	END_IF
IF  P00_PackML.fbbRecipeLoading.bOut AND GVL.bDispencer2Enable	THEN	bDispencer2EnableDelay	:= 	TRUE;	END_IF
IF  P00_PackML.fbbRecipeLoading.bOut AND GVL.bDispencer3Enable	THEN	bDispencer3EnableDelay	:= 	TRUE;	END_IF
IF  P00_PackML.fbbRecipeLoading.bOut AND GVL.bDispencer4Enable	THEN	bDispencer4EnableDelay	:= 	TRUE;	END_IF
IF NOT P00_PackML.fbbRecipeLoading.bOut THEN
	bDispencer1EnableDelay	:= FALSE;
	bDispencer2EnableDelay	:= FALSE;
	bDispencer3EnableDelay	:= FALSE;	
	bDispencer4EnableDelay	:= FALSE;	
END_IF
// Koniec podtrzymanie przy zmianie receptury






(********KASOWANIE ROZKAZÓW CYKLI*********)
IF fbDispencer1.bCycleDone AND bManualMode THEN
	VIS.bDispencer1Dose := FALSE;
END_IF
IF fbDispencer2.bCycleDone AND bManualMode THEN
	VIS.bDispencer2Dose := FALSE;
END_IF
IF fbDispencer3.bCycleDone AND bManualMode THEN
	VIS.bDispencer3Dose := FALSE;
END_IF
IF fbDispencer4.bCycleDone AND bManualMode THEN
	VIS.bDispencer4Dose := FALSE;
END_IF
 
(*****KONIEC KASOWANIA ROZKAZÓW CYKLI*****)
tonResetCloseCalibration(IN:= VIS.bDispencersCatchCloseCalibration, PT:= T#3S);
tonResetOpenCalibration	(IN:= VIS.bDispencersCatchOpenCalibration, PT:= T#3S);
IF tonResetOpenCalibration.Q THEN
	VIS.bDispencersCatchOpenCalibration	:= FALSE;
END_IF
IF tonResetCloseCalibration.Q THEN
	VIS.bDispencersCatchCloseCalibration := FALSE;
END_IF


tofDispencersDragLeftStationEnable	(IN:= GVL.bFormsDragingLeftEnable OR bFormsDragingLeftEnableDelay, 		PT:= T#10S);
tofDispencersDragRightStationEnable	(IN:= GVL.bFormsDragingRightEnable OR bFormsDragingRightEnableDelay,	PT:= T#10S);
// Dodatkowe podtrzymanie przy zmianie receptury
IF  P00_PackML.fbbRecipeLoading.bOut AND GVL.bFormsDragingLeftEnable	THEN	bFormsDragingLeftEnableDelay	:= 	TRUE;	END_IF
IF  P00_PackML.fbbRecipeLoading.bOut AND GVL.bFormsDragingRightEnable	THEN	bFormsDragingRightEnableDelay	:= 	TRUE;	END_IF
IF NOT P00_PackML.fbbRecipeLoading.bOut THEN
	bFormsDragingLeftEnableDelay	:= FALSE;
	bFormsDragingRightEnableDelay	:= FALSE;
END_IF
// Koniec podtrzymanie przy zmianie receptury


IF fbDispencersDragLeftStation.bCycleDone AND bManualMode THEN
	VIS.bFormsDragingLeftRun 									:= FALSE;
	GVL.bFormsDragingLeftPrepareRun								:= FALSE;
END_IF
IF fbDispencersDragRightStation.bCycleDone AND bManualMode THEN
	VIS.bFormsDragingRightRun 									:= FALSE;
	GVL.bFormsDragingRightPrepareRun							:= FALSE;
END_IF

ACTION aAntyColision:

//Pozycja MIN dla dozowników
IF VIS.lrDispencersCatchHeightCV-200 > 40 THEN
	fbDispencer1.lrMinPosition :=	VIS.lrDispencersCatchHeightCV-200;
	fbDispencer2.lrMinPosition :=	VIS.lrDispencersCatchHeightCV-200;
	fbDispencer3.lrMinPosition :=	VIS.lrDispencersCatchHeightCV-200;
	fbDispencer4.lrMinPosition :=	VIS.lrDispencersCatchHeightCV-200;
ELSE
	fbDispencer1.lrMinPosition :=	40;
END_IF

//Pozycja MAX dla chwytaka
IF VIS.lrDispencer12LifterActPos < VIS.lrDispencer34LifterActPos THEN
	fbDispencersCatch1Station.lrMaxHeight := VIS.lrDispencer12LifterActPos + 200;
ELSE
	fbDispencersCatch1Station.lrMaxHeight := VIS.lrDispencer34LifterActPos + 200;
END_IF
END_ACTION

ACTION aCleaning:
(*** MYCIE DOZOWNIKÓW CIP 12***)
(* Doza naprzemienna i pompowanie zbiornika*)

//Zmienne
VIS.bDispencersCIP;		//Włączony CIP z wizu
bCIP;					//Przefiltrowany sygnał CIP
VIS.iDispencersCIP;		//Informacja o ruchu wylewek
VIS.bDispencer12Cleaning;
VIS.bDispencer34Cleaning;
eDispencer1RunningState;		aDispencer1AxisRef.NcToPlc.ActPos;
eDispencer2RunningState;		aDispencer2AxisRef.NcToPlc.ActPos;
VIS.bDispencer12Cleaning;		bDispencer1Cleaning;bDispencer2Cleaning;
VIS.lrDispencersManualOverride;


//Filtrowanie sygnału, przeciw lagom z wizualizacji lub ciągłym klikaniem
fbDispencersCIP(bIn:=VIS.bDispencersCIP,tFilterTimeOn:=T#0MS,tFilterTimeOff:=T#3S,bOUT=>bCIP);

tonbCIP	(IN:=bCIP, PT:=T#7S);
ftbCIP	(CLK:=bCIP,	Q=>);
rtbCIP	(CLK:=bCIP,	Q=>);

IF rtbCIP.Q THEN
	VIS.bTank1SupplyPumpEnableShow:=FALSE;
	VIS.bTank2SupplyPumpEnableShow:=FALSE;
END_IF

//Przejazd chwytaków i dozowników
IF bCIP THEN
	VIS.bDispencer12ManualLifterDown	:= VIS.lrDispencer12LifterActPos	>	40;
	VIS.bDispencer34ManualLifterDown	:= VIS.lrDispencer34LifterActPos	>	40;
	VIS.iDispencersCIP := 0;
	IF tonbCIP.Q THEN // Ustawianie informacji o stacji z opóźnieniem
		IF P02_Dispencers.fbDispencersCatch1Station.eState = E_Station.ePreparingToDisable OR P02_Dispencers.fbDispencersCatch1Station.eState = E_Station.eHoming
		OR VIS.bDispencer12ManualLifterDown OR VIS.bDispencer34ManualLifterDown
		THEN
			VIS.iDispencersCIP 			:=	0;
		ELSIF P02_Dispencers.fbDispencersCatch1Station.eState = E_Station.eDisabled THEN
			VIS.iDispencersCIP 			:=	-1;
		END_IF 
	END_IF
END_IF

//Kasowanie rozkazów na wszelki wypadek
IF ftbCIP.Q THEN
	VIS.bDispencer12ManualLifterDown 		:= FALSE;
	VIS.bDispencer34ManualLifterDown 		:= FALSE;
	VIS.bDispencer1ManualSuckValve			:= FALSE;
	VIS.bDispencer1ManualDoseValve			:= FALSE;
	VIS.bDispencer2ManualSuckValve			:= FALSE;
	VIS.bDispencer2ManualDoseValve			:= FALSE;
	VIS.bDispencer3ManualSuckValve			:= FALSE;
	VIS.bDispencer3ManualDoseValve			:= FALSE;
	VIS.bDispencer4ManualSuckValve			:= FALSE;
	VIS.bDispencer4ManualDoseValve			:= FALSE;
	VIS.iDispencersCIP := 0;
END_IF


//PID regulacji poziomu
fbDispencersCleaningPID(
	bEnable:= VIS.bDispencer12Cleaning OR VIS.bDispencer34Cleaning , 
	bInvertDirection:=TRUE , 
	lrSetpointValue:= 20, 
	lrActualValue:= iTank1Sensor1Value, 
	bReset:= , 
	lrYMin:= 50, 
	lrYMax:= 100, 
	lrKp:= 0.0001, 
	tTn:= T#10S, 
	tTv:= , 
	tTd:=T#0S , 
	lrTaskCycleTime:=10.0 , 
	lrCycleTime:= 1000, 
	lrY=> , 
	bError=> );
 
//Wyłączenie mycia CIP po czasie	
tonbDispencer12Cleaning(IN:=VIS.bDispencer12Cleaning, PT:=T#360S);
IF tonbDispencer12Cleaning.Q THEN
	VIS.bDispencer12Cleaning := FALSE;
END_IF
tonbDispencer34Cleaning(IN:=VIS.bDispencer34Cleaning, PT:=T#360S);
IF tonbDispencer34Cleaning.Q THEN
	VIS.bDispencer34Cleaning := FALSE;
END_IF


IF VIS.bTank1ManualSupplyPump AND VIS.bTank1LevelSensorHigh AND VIS.iTank1LevelSensorValue>110 THEN
	VIS.bTank1ManualSupplyPump := FALSE;
END_IF

//DOZOWNIKI 1 i 2 | Procedura mycia CIP
IF VIS.bDispencer12Cleaning THEN
	//Ustawienie njaniższego poziomu w zbiorniku
	VIS.uTank1LevelSetpointShow;VIS.bTank1LevelSensorLow;VIS.bTank1LevelSensorHigh; //Ustawianie w aTanks
	//Włączenie pompy
	VIS.bTank1SupplyPumpEnableShow;VIS.bTank1ManualSupplyPump;
	//Ustawienie override od PIDa
	//VIS.lrDispencerManualOverride	:= fbDispencersCleaningPID.lrY; 
	//Dozownaie naprzemienne
	IF eDispencer1RunningState = E_DispencerState.eCleaningReady  THEN
	 	bDispencer1Cleaning 		:=	TRUE;
	END_IF	
	IF eDispencer2RunningState = E_DispencerState.eCleaningReady  AND (eDispencer1RunningState = E_DispencerState.eCleaning AND aDispencer1AxisRef.NcToPlc.ActPos < 100) THEN
		bDispencer2Cleaning 		:=	TRUE;
	END_IF
	IF eDispencer1RunningState = E_DispencerState.eCleaningDone  THEN
	 	bDispencer1Cleaning 		:=	FALSE;
	END_IF
	IF eDispencer2RunningState = E_DispencerState.eCleaningDone  THEN
	 	bDispencer2Cleaning 		:=	FALSE;
	END_IF		
ELSE //Czyszczenie 
	 bDispencer1Cleaning			:= bDispencer2Cleaning	:=	FALSE;
END_IF

//DOZOWNIKI 3 i 4 | Procedura mycia CIP
IF VIS.bDispencer34Cleaning THEN
	//Ustawienie njaniższego poziomu w zbiorniku
	VIS.uTank1LevelSetpointShow;VIS.bTank1LevelSensorLow;VIS.bTank1LevelSensorHigh; //Ustawianie w aTanks
	//Ustawienie override od PIDa
	//VIS.lrDispencerManualOverride	:= fbDispencersCleaningPID.lrY; 
	//Dozownaie naprzemienne
	IF eDispencer3RunningState = E_DispencerState.eCleaningReady  THEN
	 	bDispencer3Cleaning 		:=	TRUE;
	END_IF	
	IF eDispencer4RunningState = E_DispencerState.eCleaningReady  AND (eDispencer3RunningState = E_DispencerState.eCleaning AND aDispencer3AxisRef.NcToPlc.ActPos < 100) THEN
		bDispencer4Cleaning 		:=	TRUE;
	END_IF
	IF eDispencer3RunningState = E_DispencerState.eCleaningDone  THEN
	 	bDispencer3Cleaning 		:=	FALSE;
	END_IF
	IF eDispencer4RunningState = E_DispencerState.eCleaningDone  THEN
	 	bDispencer4Cleaning 		:=	FALSE;
	END_IF		
	 
ELSE //Czyszczenie 
	 bDispencer3Cleaning			:= bDispencer4Cleaning	:=	FALSE;
END_IF
		
// WYłączanie pompy
IF NOT VIS.bDispencer12Cleaning AND NOT VIS.bDispencer34Cleaning THEN
	VIS.lrDispencersManualOverride := 100;
END_IF
END_ACTION

ACTION aDispencer1:
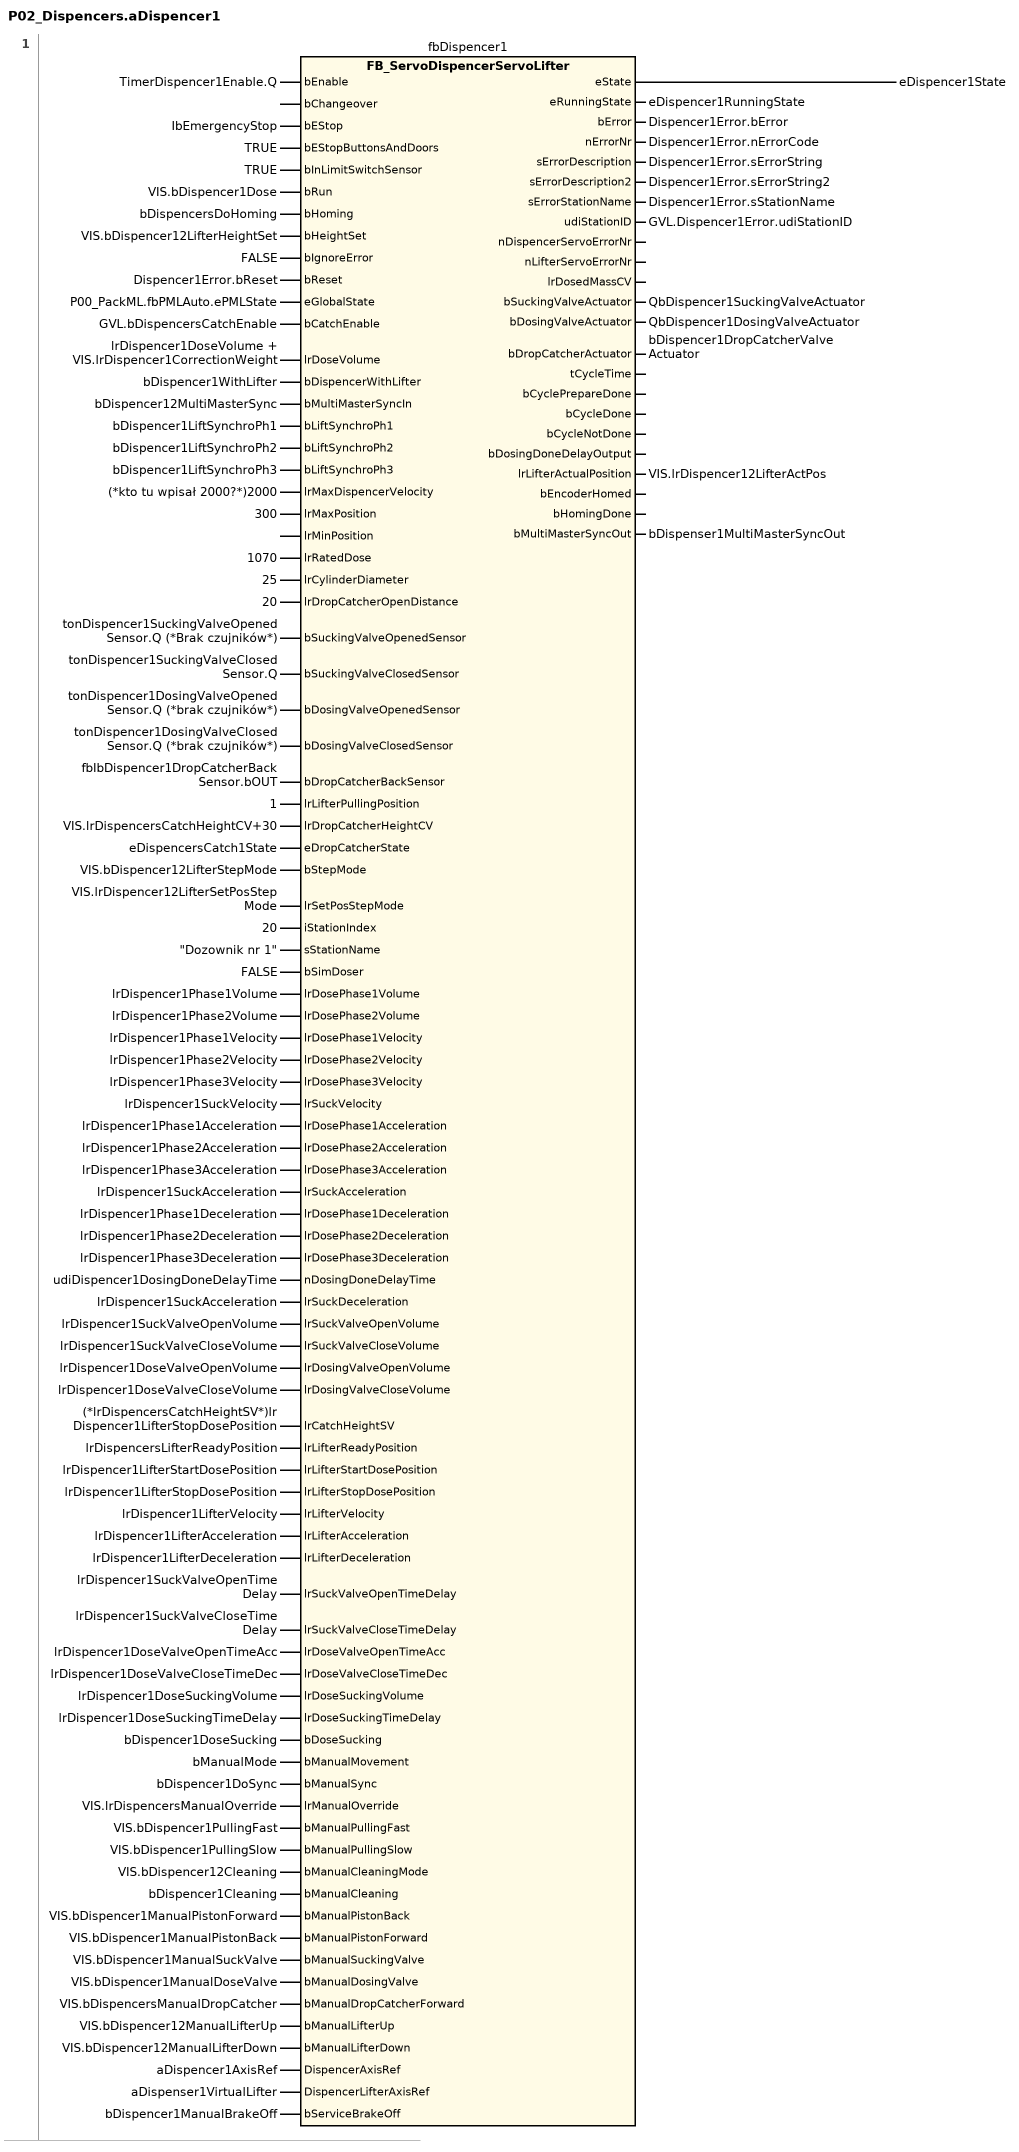
// NETWORK 1
fbDispencer1(
    bEnable := TimerDispencer1Enable.Q,
    bEStop := IbEmergencyStop,
    bEStopButtonsAndDoors := TRUE,
    bInLimitSwitchSensor := TRUE,
    bRun := VIS.bDispencer1Dose,
    bHoming := bDispencersDoHoming,
    bHeightSet := VIS.bDispencer12LifterHeightSet,
    bIgnoreError := FALSE,
    bReset := Dispencer1Error.bReset,
    eGlobalState := P00_PackML.fbPMLAuto.ePMLState,
    bCatchEnable := GVL.bDispencersCatchEnable,
    lrDoseVolume := lrDispencer1DoseVolume + VIS.lrDispencer1CorrectionWeight,
    bDispencerWithLifter := bDispencer1WithLifter,
    bMultiMasterSyncIn := bDispencer12MultiMasterSync,
    bLiftSynchroPh1 := bDispencer1LiftSynchroPh1,
    bLiftSynchroPh2 := bDispencer1LiftSynchroPh2,
    bLiftSynchroPh3 := bDispencer1LiftSynchroPh3,
    lrMaxDispencerVelocity := (*kto tu wpisał 2000?*)2000,
    lrMaxPosition := 300,
    lrRatedDose := 1070,
    lrCylinderDiameter := 25,
    lrDropCatcherOpenDistance := 20,
    bSuckingValveOpenedSensor := tonDispencer1SuckingValveOpenedSensor.Q (*Brak czujników*),
    bSuckingValveClosedSensor := tonDispencer1SuckingValveClosedSensor.Q,
    bDosingValveOpenedSensor := tonDispencer1DosingValveOpenedSensor.Q (*brak czujników*),
    bDosingValveClosedSensor := tonDispencer1DosingValveClosedSensor.Q (*brak czujników*),
    bDropCatcherBackSensor := fbIbDispencer1DropCatcherBackSensor.bOUT,
    lrLifterPullingPosition := 1,
    lrDropCatcherHeightCV := VIS.lrDispencersCatchHeightCV+30,
    eDropCatcherState := eDispencersCatch1State,
    bStepMode := VIS.bDispencer12LifterStepMode,
    lrSetPosStepMode := VIS.lrDispencer12LifterSetPosStepMode,
    iStationIndex := 20,
    sStationName := "Dozownik nr 1",
    bSimDoser := FALSE,
    lrDosePhase1Volume := lrDispencer1Phase1Volume,
    lrDosePhase2Volume := lrDispencer1Phase2Volume,
    lrDosePhase1Velocity := lrDispencer1Phase1Velocity,
    lrDosePhase2Velocity := lrDispencer1Phase2Velocity,
    lrDosePhase3Velocity := lrDispencer1Phase3Velocity,
    lrSuckVelocity := lrDispencer1SuckVelocity,
    lrDosePhase1Acceleration := lrDispencer1Phase1Acceleration,
    lrDosePhase2Acceleration := lrDispencer1Phase2Acceleration,
    lrDosePhase3Acceleration := lrDispencer1Phase3Acceleration,
    lrSuckAcceleration := lrDispencer1SuckAcceleration,
    lrDosePhase1Deceleration := lrDispencer1Phase1Deceleration,
    lrDosePhase2Deceleration := lrDispencer1Phase2Deceleration,
    lrDosePhase3Deceleration := lrDispencer1Phase3Deceleration,
    nDosingDoneDelayTime := udiDispencer1DosingDoneDelayTime,
    lrSuckDeceleration := lrDispencer1SuckAcceleration,
    lrSuckValveOpenVolume := lrDispencer1SuckValveOpenVolume,
    lrSuckValveCloseVolume := lrDispencer1SuckValveCloseVolume,
    lrDosingValveOpenVolume := lrDispencer1DoseValveOpenVolume,
    lrDosingValveCloseVolume := lrDispencer1DoseValveCloseVolume,
    lrCatchHeightSV := (*lrDispencersCatchHeightSV*)lrDispencer1LifterStopDosePosition,
    lrLifterReadyPosition := lrDispencersLifterReadyPosition,
    lrLifterStartDosePosition := lrDispencer1LifterStartDosePosition,
    lrLifterStopDosePosition := lrDispencer1LifterStopDosePosition,
    lrLifterVelocity := lrDispencer1LifterVelocity,
    lrLifterAcceleration := lrDispencer1LifterAcceleration,
    lrLifterDeceleration := lrDispencer1LifterDeceleration,
    lrSuckValveOpenTimeDelay := lrDispencer1SuckValveOpenTimeDelay,
    lrSuckValveCloseTimeDelay := lrDispencer1SuckValveCloseTimeDelay,
    lrDoseValveOpenTimeAcc := lrDispencer1DoseValveOpenTimeAcc,
    lrDoseValveCloseTimeDec := lrDispencer1DoseValveCloseTimeDec,
    lrDoseSuckingVolume := lrDispencer1DoseSuckingVolume,
    lrDoseSuckingTimeDelay := lrDispencer1DoseSuckingTimeDelay,
    bDoseSucking := bDispencer1DoseSucking,
    bManualMovement := bManualMode,
    bManualSync := bDispencer1DoSync,
    lrManualOverride := VIS.lrDispencersManualOverride,
    bManualPullingFast := VIS.bDispencer1PullingFast,
    bManualPullingSlow := VIS.bDispencer1PullingSlow,
    bManualCleaningMode := VIS.bDispencer12Cleaning,
    bManualCleaning := bDispencer1Cleaning,
    bManualPistonBack := VIS.bDispencer1ManualPistonForward,
    bManualPistonForward := VIS.bDispencer1ManualPistonBack,
    bManualSuckingValve := VIS.bDispencer1ManualSuckValve,
    bManualDosingValve := VIS.bDispencer1ManualDoseValve,
    bManualDropCatcherForward := VIS.bDispencersManualDropCatcher,
    bManualLifterUp := VIS.bDispencer12ManualLifterUp,
    bManualLifterDown := VIS.bDispencer12ManualLifterDown,
    DispencerAxisRef := aDispencer1AxisRef,
    DispencerLifterAxisRef := aDispenser1VirtualLifter,
    bServiceBrakeOff := bDispencer1ManualBrakeOff,
    eRunningState => eDispencer1RunningState,
    bError => Dispencer1Error.bError,
    nErrorNr => Dispencer1Error.nErrorCode,
    sErrorDescription => Dispencer1Error.sErrorString,
    sErrorDescription2 => Dispencer1Error.sErrorString2,
    sErrorStationName => Dispencer1Error.sStationName,
    udiStationID => GVL.Dispencer1Error.udiStationID,
    bSuckingValveActuator => QbDispencer1SuckingValveActuator,
    bDosingValveActuator => QbDispencer1DosingValveActuator,
    bDropCatcherActuator => bDispencer1DropCatcherValveActuator,
    lrLifterActualPosition => VIS.lrDispencer12LifterActPos,
    bMultiMasterSyncOut => bDispenser1MultiMasterSyncOut); // FB_ServoDispencerServoLifter
eDispencer1State := fbDispencer1.eState;
END_ACTION

ACTION aDispencer2:
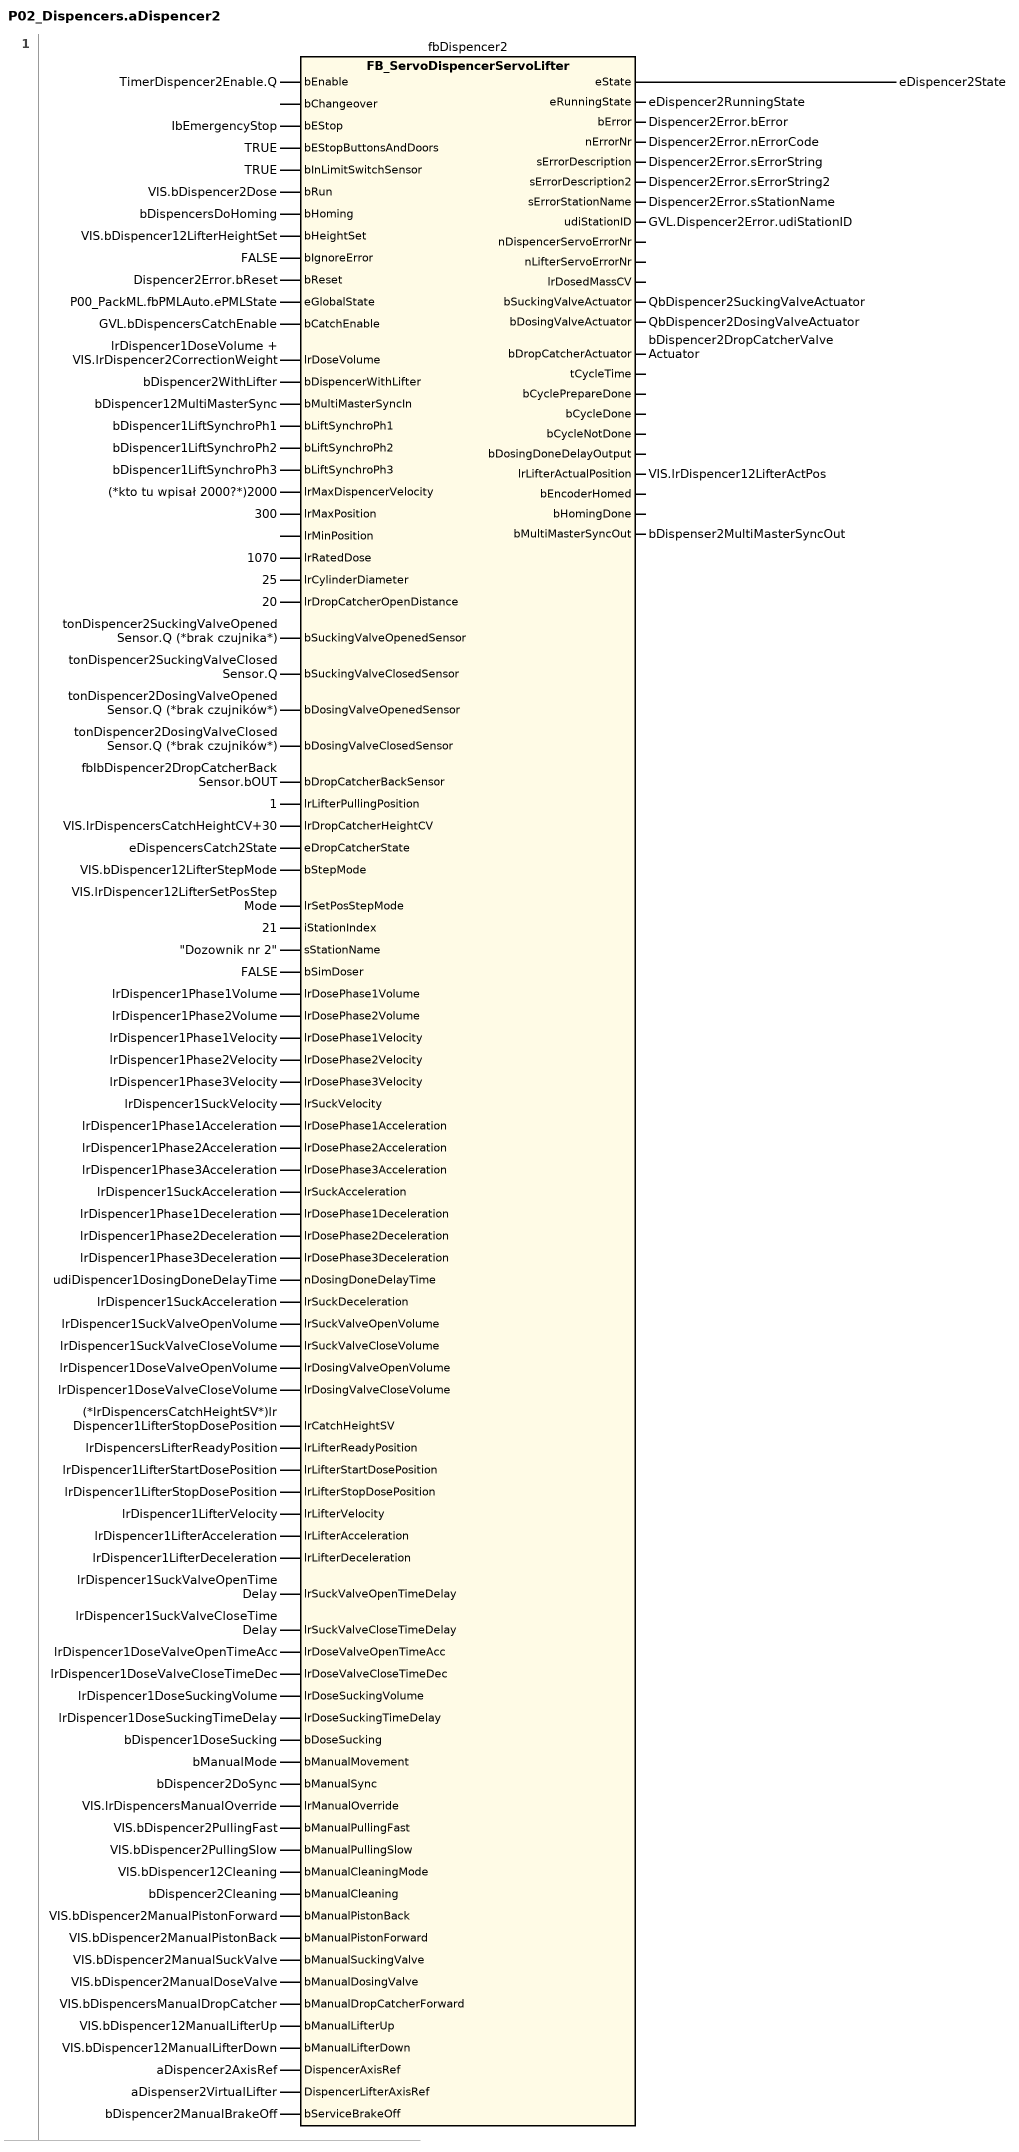
// NETWORK 1
fbDispencer2(
    bEnable := TimerDispencer2Enable.Q,
    bEStop := IbEmergencyStop,
    bEStopButtonsAndDoors := TRUE,
    bInLimitSwitchSensor := TRUE,
    bRun := VIS.bDispencer2Dose,
    bHoming := bDispencersDoHoming,
    bHeightSet := VIS.bDispencer12LifterHeightSet,
    bIgnoreError := FALSE,
    bReset := Dispencer2Error.bReset,
    eGlobalState := P00_PackML.fbPMLAuto.ePMLState,
    bCatchEnable := GVL.bDispencersCatchEnable,
    lrDoseVolume := lrDispencer1DoseVolume + VIS.lrDispencer2CorrectionWeight,
    bDispencerWithLifter := bDispencer2WithLifter,
    bMultiMasterSyncIn := bDispencer12MultiMasterSync,
    bLiftSynchroPh1 := bDispencer1LiftSynchroPh1,
    bLiftSynchroPh2 := bDispencer1LiftSynchroPh2,
    bLiftSynchroPh3 := bDispencer1LiftSynchroPh3,
    lrMaxDispencerVelocity := (*kto tu wpisał 2000?*)2000,
    lrMaxPosition := 300,
    lrRatedDose := 1070,
    lrCylinderDiameter := 25,
    lrDropCatcherOpenDistance := 20,
    bSuckingValveOpenedSensor := tonDispencer2SuckingValveOpenedSensor.Q (*brak czujnika*),
    bSuckingValveClosedSensor := tonDispencer2SuckingValveClosedSensor.Q,
    bDosingValveOpenedSensor := tonDispencer2DosingValveOpenedSensor.Q (*brak czujników*),
    bDosingValveClosedSensor := tonDispencer2DosingValveClosedSensor.Q (*brak czujników*),
    bDropCatcherBackSensor := fbIbDispencer2DropCatcherBackSensor.bOUT,
    lrLifterPullingPosition := 1,
    lrDropCatcherHeightCV := VIS.lrDispencersCatchHeightCV+30,
    eDropCatcherState := eDispencersCatch2State,
    bStepMode := VIS.bDispencer12LifterStepMode,
    lrSetPosStepMode := VIS.lrDispencer12LifterSetPosStepMode,
    iStationIndex := 21,
    sStationName := "Dozownik nr 2",
    bSimDoser := FALSE,
    lrDosePhase1Volume := lrDispencer1Phase1Volume,
    lrDosePhase2Volume := lrDispencer1Phase2Volume,
    lrDosePhase1Velocity := lrDispencer1Phase1Velocity,
    lrDosePhase2Velocity := lrDispencer1Phase2Velocity,
    lrDosePhase3Velocity := lrDispencer1Phase3Velocity,
    lrSuckVelocity := lrDispencer1SuckVelocity,
    lrDosePhase1Acceleration := lrDispencer1Phase1Acceleration,
    lrDosePhase2Acceleration := lrDispencer1Phase2Acceleration,
    lrDosePhase3Acceleration := lrDispencer1Phase3Acceleration,
    lrSuckAcceleration := lrDispencer1SuckAcceleration,
    lrDosePhase1Deceleration := lrDispencer1Phase1Deceleration,
    lrDosePhase2Deceleration := lrDispencer1Phase2Deceleration,
    lrDosePhase3Deceleration := lrDispencer1Phase3Deceleration,
    nDosingDoneDelayTime := udiDispencer1DosingDoneDelayTime,
    lrSuckDeceleration := lrDispencer1SuckAcceleration,
    lrSuckValveOpenVolume := lrDispencer1SuckValveOpenVolume,
    lrSuckValveCloseVolume := lrDispencer1SuckValveCloseVolume,
    lrDosingValveOpenVolume := lrDispencer1DoseValveOpenVolume,
    lrDosingValveCloseVolume := lrDispencer1DoseValveCloseVolume,
    lrCatchHeightSV := (*lrDispencersCatchHeightSV*)lrDispencer1LifterStopDosePosition,
    lrLifterReadyPosition := lrDispencersLifterReadyPosition,
    lrLifterStartDosePosition := lrDispencer1LifterStartDosePosition,
    lrLifterStopDosePosition := lrDispencer1LifterStopDosePosition,
    lrLifterVelocity := lrDispencer1LifterVelocity,
    lrLifterAcceleration := lrDispencer1LifterAcceleration,
    lrLifterDeceleration := lrDispencer1LifterDeceleration,
    lrSuckValveOpenTimeDelay := lrDispencer1SuckValveOpenTimeDelay,
    lrSuckValveCloseTimeDelay := lrDispencer1SuckValveCloseTimeDelay,
    lrDoseValveOpenTimeAcc := lrDispencer1DoseValveOpenTimeAcc,
    lrDoseValveCloseTimeDec := lrDispencer1DoseValveCloseTimeDec,
    lrDoseSuckingVolume := lrDispencer1DoseSuckingVolume,
    lrDoseSuckingTimeDelay := lrDispencer1DoseSuckingTimeDelay,
    bDoseSucking := bDispencer1DoseSucking,
    bManualMovement := bManualMode,
    bManualSync := bDispencer2DoSync,
    lrManualOverride := VIS.lrDispencersManualOverride,
    bManualPullingFast := VIS.bDispencer2PullingFast,
    bManualPullingSlow := VIS.bDispencer2PullingSlow,
    bManualCleaningMode := VIS.bDispencer12Cleaning,
    bManualCleaning := bDispencer2Cleaning,
    bManualPistonBack := VIS.bDispencer2ManualPistonForward,
    bManualPistonForward := VIS.bDispencer2ManualPistonBack,
    bManualSuckingValve := VIS.bDispencer2ManualSuckValve,
    bManualDosingValve := VIS.bDispencer2ManualDoseValve,
    bManualDropCatcherForward := VIS.bDispencersManualDropCatcher,
    bManualLifterUp := VIS.bDispencer12ManualLifterUp,
    bManualLifterDown := VIS.bDispencer12ManualLifterDown,
    DispencerAxisRef := aDispencer2AxisRef,
    DispencerLifterAxisRef := aDispenser2VirtualLifter,
    bServiceBrakeOff := bDispencer2ManualBrakeOff,
    eRunningState => eDispencer2RunningState,
    bError => Dispencer2Error.bError,
    nErrorNr => Dispencer2Error.nErrorCode,
    sErrorDescription => Dispencer2Error.sErrorString,
    sErrorDescription2 => Dispencer2Error.sErrorString2,
    sErrorStationName => Dispencer2Error.sStationName,
    udiStationID => GVL.Dispencer2Error.udiStationID,
    bSuckingValveActuator => QbDispencer2SuckingValveActuator,
    bDosingValveActuator => QbDispencer2DosingValveActuator,
    bDropCatcherActuator => bDispencer2DropCatcherValveActuator,
    lrLifterActualPosition => VIS.lrDispencer12LifterActPos,
    bMultiMasterSyncOut => bDispenser2MultiMasterSyncOut); // FB_ServoDispencerServoLifter
eDispencer2State := fbDispencer2.eState;
END_ACTION

ACTION aDispencer3:
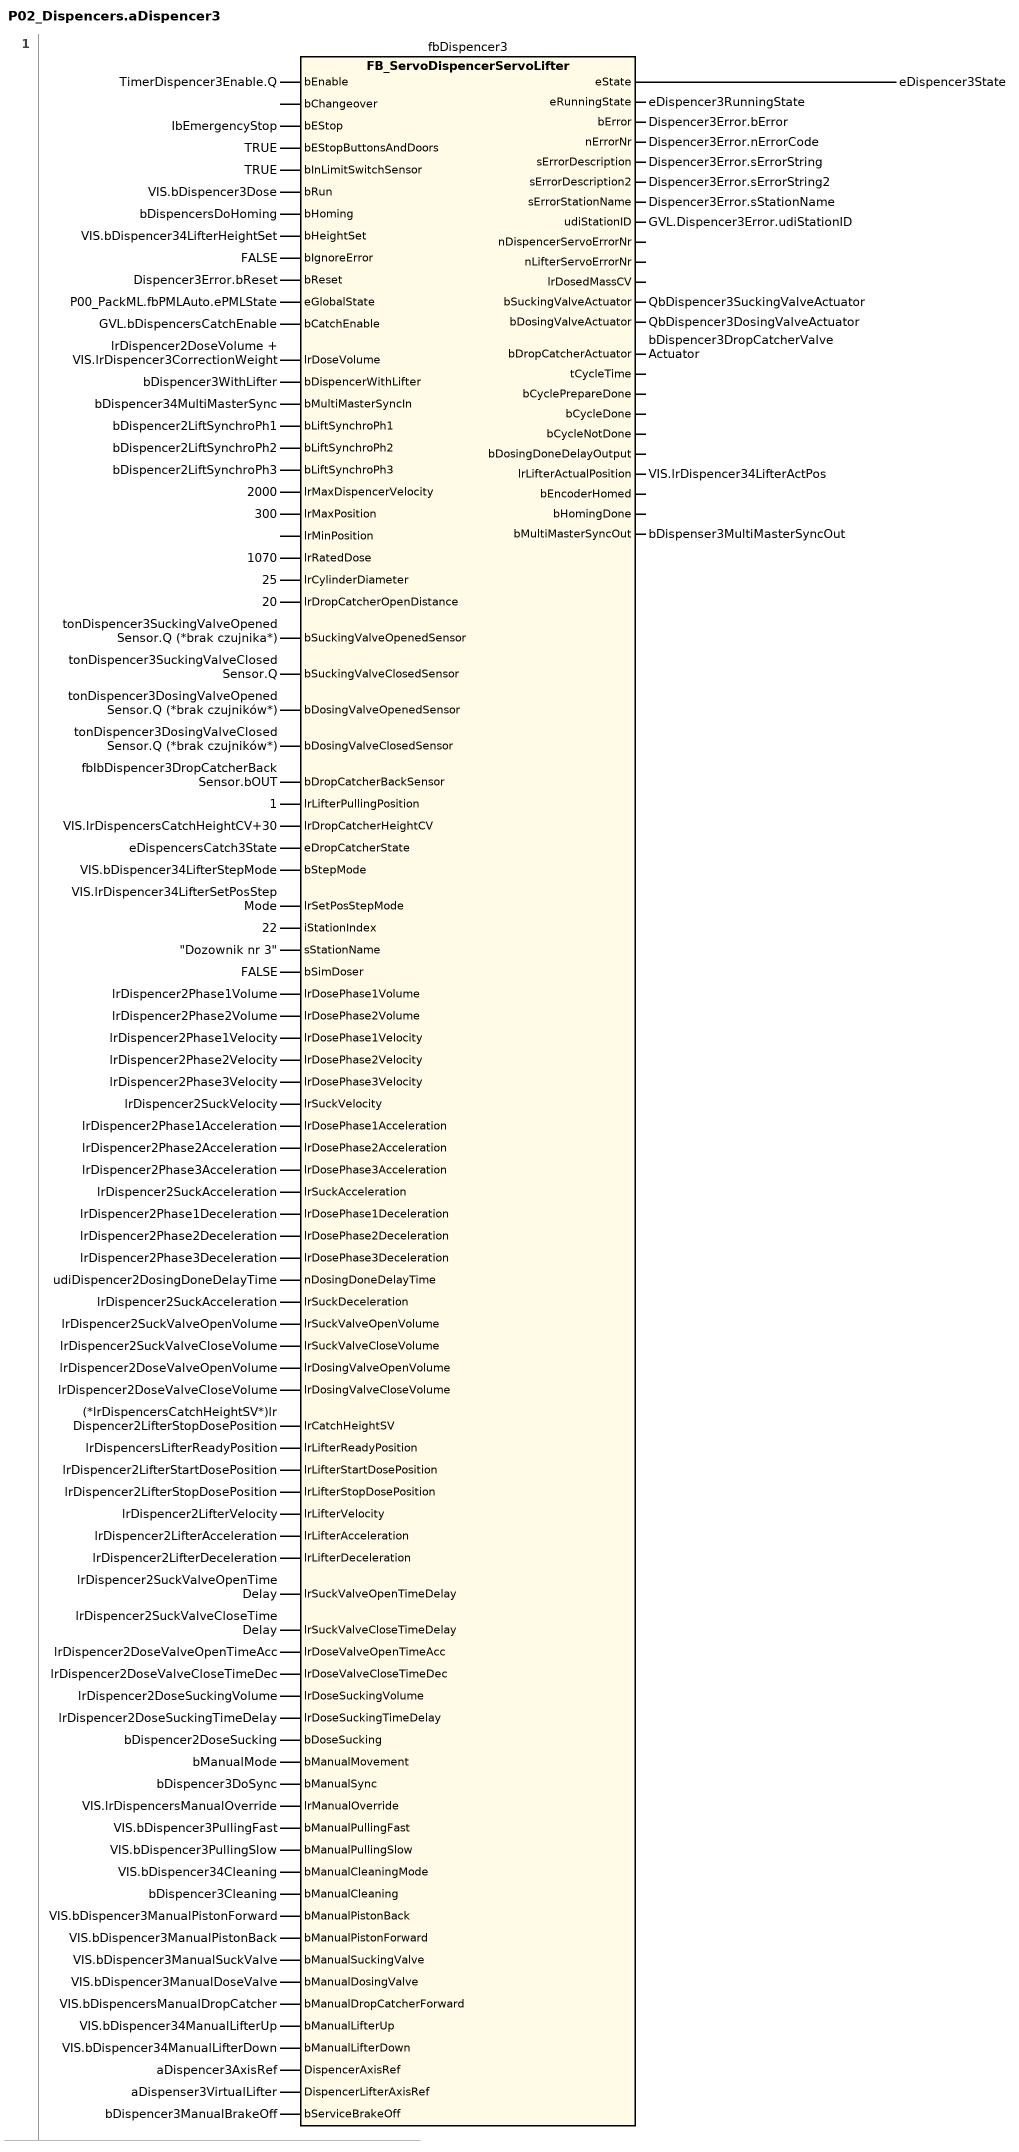
// NETWORK 1
fbDispencer3(
    bEnable := TimerDispencer3Enable.Q,
    bEStop := IbEmergencyStop,
    bEStopButtonsAndDoors := TRUE,
    bInLimitSwitchSensor := TRUE,
    bRun := VIS.bDispencer3Dose,
    bHoming := bDispencersDoHoming,
    bHeightSet := VIS.bDispencer34LifterHeightSet,
    bIgnoreError := FALSE,
    bReset := Dispencer3Error.bReset,
    eGlobalState := P00_PackML.fbPMLAuto.ePMLState,
    bCatchEnable := GVL.bDispencersCatchEnable,
    lrDoseVolume := lrDispencer2DoseVolume + VIS.lrDispencer3CorrectionWeight,
    bDispencerWithLifter := bDispencer3WithLifter,
    bMultiMasterSyncIn := bDispencer34MultiMasterSync,
    bLiftSynchroPh1 := bDispencer2LiftSynchroPh1,
    bLiftSynchroPh2 := bDispencer2LiftSynchroPh2,
    bLiftSynchroPh3 := bDispencer2LiftSynchroPh3,
    lrMaxDispencerVelocity := 2000,
    lrMaxPosition := 300,
    lrRatedDose := 1070,
    lrCylinderDiameter := 25,
    lrDropCatcherOpenDistance := 20,
    bSuckingValveOpenedSensor := tonDispencer3SuckingValveOpenedSensor.Q (*brak czujnika*),
    bSuckingValveClosedSensor := tonDispencer3SuckingValveClosedSensor.Q,
    bDosingValveOpenedSensor := tonDispencer3DosingValveOpenedSensor.Q (*brak czujników*),
    bDosingValveClosedSensor := tonDispencer3DosingValveClosedSensor.Q (*brak czujników*),
    bDropCatcherBackSensor := fbIbDispencer3DropCatcherBackSensor.bOUT,
    lrLifterPullingPosition := 1,
    lrDropCatcherHeightCV := VIS.lrDispencersCatchHeightCV+30,
    eDropCatcherState := eDispencersCatch3State,
    bStepMode := VIS.bDispencer34LifterStepMode,
    lrSetPosStepMode := VIS.lrDispencer34LifterSetPosStepMode,
    iStationIndex := 22,
    sStationName := "Dozownik nr 3",
    bSimDoser := FALSE,
    lrDosePhase1Volume := lrDispencer2Phase1Volume,
    lrDosePhase2Volume := lrDispencer2Phase2Volume,
    lrDosePhase1Velocity := lrDispencer2Phase1Velocity,
    lrDosePhase2Velocity := lrDispencer2Phase2Velocity,
    lrDosePhase3Velocity := lrDispencer2Phase3Velocity,
    lrSuckVelocity := lrDispencer2SuckVelocity,
    lrDosePhase1Acceleration := lrDispencer2Phase1Acceleration,
    lrDosePhase2Acceleration := lrDispencer2Phase2Acceleration,
    lrDosePhase3Acceleration := lrDispencer2Phase3Acceleration,
    lrSuckAcceleration := lrDispencer2SuckAcceleration,
    lrDosePhase1Deceleration := lrDispencer2Phase1Deceleration,
    lrDosePhase2Deceleration := lrDispencer2Phase2Deceleration,
    lrDosePhase3Deceleration := lrDispencer2Phase3Deceleration,
    nDosingDoneDelayTime := udiDispencer2DosingDoneDelayTime,
    lrSuckDeceleration := lrDispencer2SuckAcceleration,
    lrSuckValveOpenVolume := lrDispencer2SuckValveOpenVolume,
    lrSuckValveCloseVolume := lrDispencer2SuckValveCloseVolume,
    lrDosingValveOpenVolume := lrDispencer2DoseValveOpenVolume,
    lrDosingValveCloseVolume := lrDispencer2DoseValveCloseVolume,
    lrCatchHeightSV := (*lrDispencersCatchHeightSV*)lrDispencer2LifterStopDosePosition,
    lrLifterReadyPosition := lrDispencersLifterReadyPosition,
    lrLifterStartDosePosition := lrDispencer2LifterStartDosePosition,
    lrLifterStopDosePosition := lrDispencer2LifterStopDosePosition,
    lrLifterVelocity := lrDispencer2LifterVelocity,
    lrLifterAcceleration := lrDispencer2LifterAcceleration,
    lrLifterDeceleration := lrDispencer2LifterDeceleration,
    lrSuckValveOpenTimeDelay := lrDispencer2SuckValveOpenTimeDelay,
    lrSuckValveCloseTimeDelay := lrDispencer2SuckValveCloseTimeDelay,
    lrDoseValveOpenTimeAcc := lrDispencer2DoseValveOpenTimeAcc,
    lrDoseValveCloseTimeDec := lrDispencer2DoseValveCloseTimeDec,
    lrDoseSuckingVolume := lrDispencer2DoseSuckingVolume,
    lrDoseSuckingTimeDelay := lrDispencer2DoseSuckingTimeDelay,
    bDoseSucking := bDispencer2DoseSucking,
    bManualMovement := bManualMode,
    bManualSync := bDispencer3DoSync,
    lrManualOverride := VIS.lrDispencersManualOverride,
    bManualPullingFast := VIS.bDispencer3PullingFast,
    bManualPullingSlow := VIS.bDispencer3PullingSlow,
    bManualCleaningMode := VIS.bDispencer34Cleaning,
    bManualCleaning := bDispencer3Cleaning,
    bManualPistonBack := VIS.bDispencer3ManualPistonForward,
    bManualPistonForward := VIS.bDispencer3ManualPistonBack,
    bManualSuckingValve := VIS.bDispencer3ManualSuckValve,
    bManualDosingValve := VIS.bDispencer3ManualDoseValve,
    bManualDropCatcherForward := VIS.bDispencersManualDropCatcher,
    bManualLifterUp := VIS.bDispencer34ManualLifterUp,
    bManualLifterDown := VIS.bDispencer34ManualLifterDown,
    DispencerAxisRef := aDispencer3AxisRef,
    DispencerLifterAxisRef := aDispenser3VirtualLifter,
    bServiceBrakeOff := bDispencer3ManualBrakeOff,
    eRunningState => eDispencer3RunningState,
    bError => Dispencer3Error.bError,
    nErrorNr => Dispencer3Error.nErrorCode,
    sErrorDescription => Dispencer3Error.sErrorString,
    sErrorDescription2 => Dispencer3Error.sErrorString2,
    sErrorStationName => Dispencer3Error.sStationName,
    udiStationID => GVL.Dispencer3Error.udiStationID,
    bSuckingValveActuator => QbDispencer3SuckingValveActuator,
    bDosingValveActuator => QbDispencer3DosingValveActuator,
    bDropCatcherActuator => bDispencer3DropCatcherValveActuator,
    lrLifterActualPosition => VIS.lrDispencer34LifterActPos,
    bMultiMasterSyncOut => bDispenser3MultiMasterSyncOut); // FB_ServoDispencerServoLifter
eDispencer3State := fbDispencer3.eState;
END_ACTION

ACTION aDispencer4:
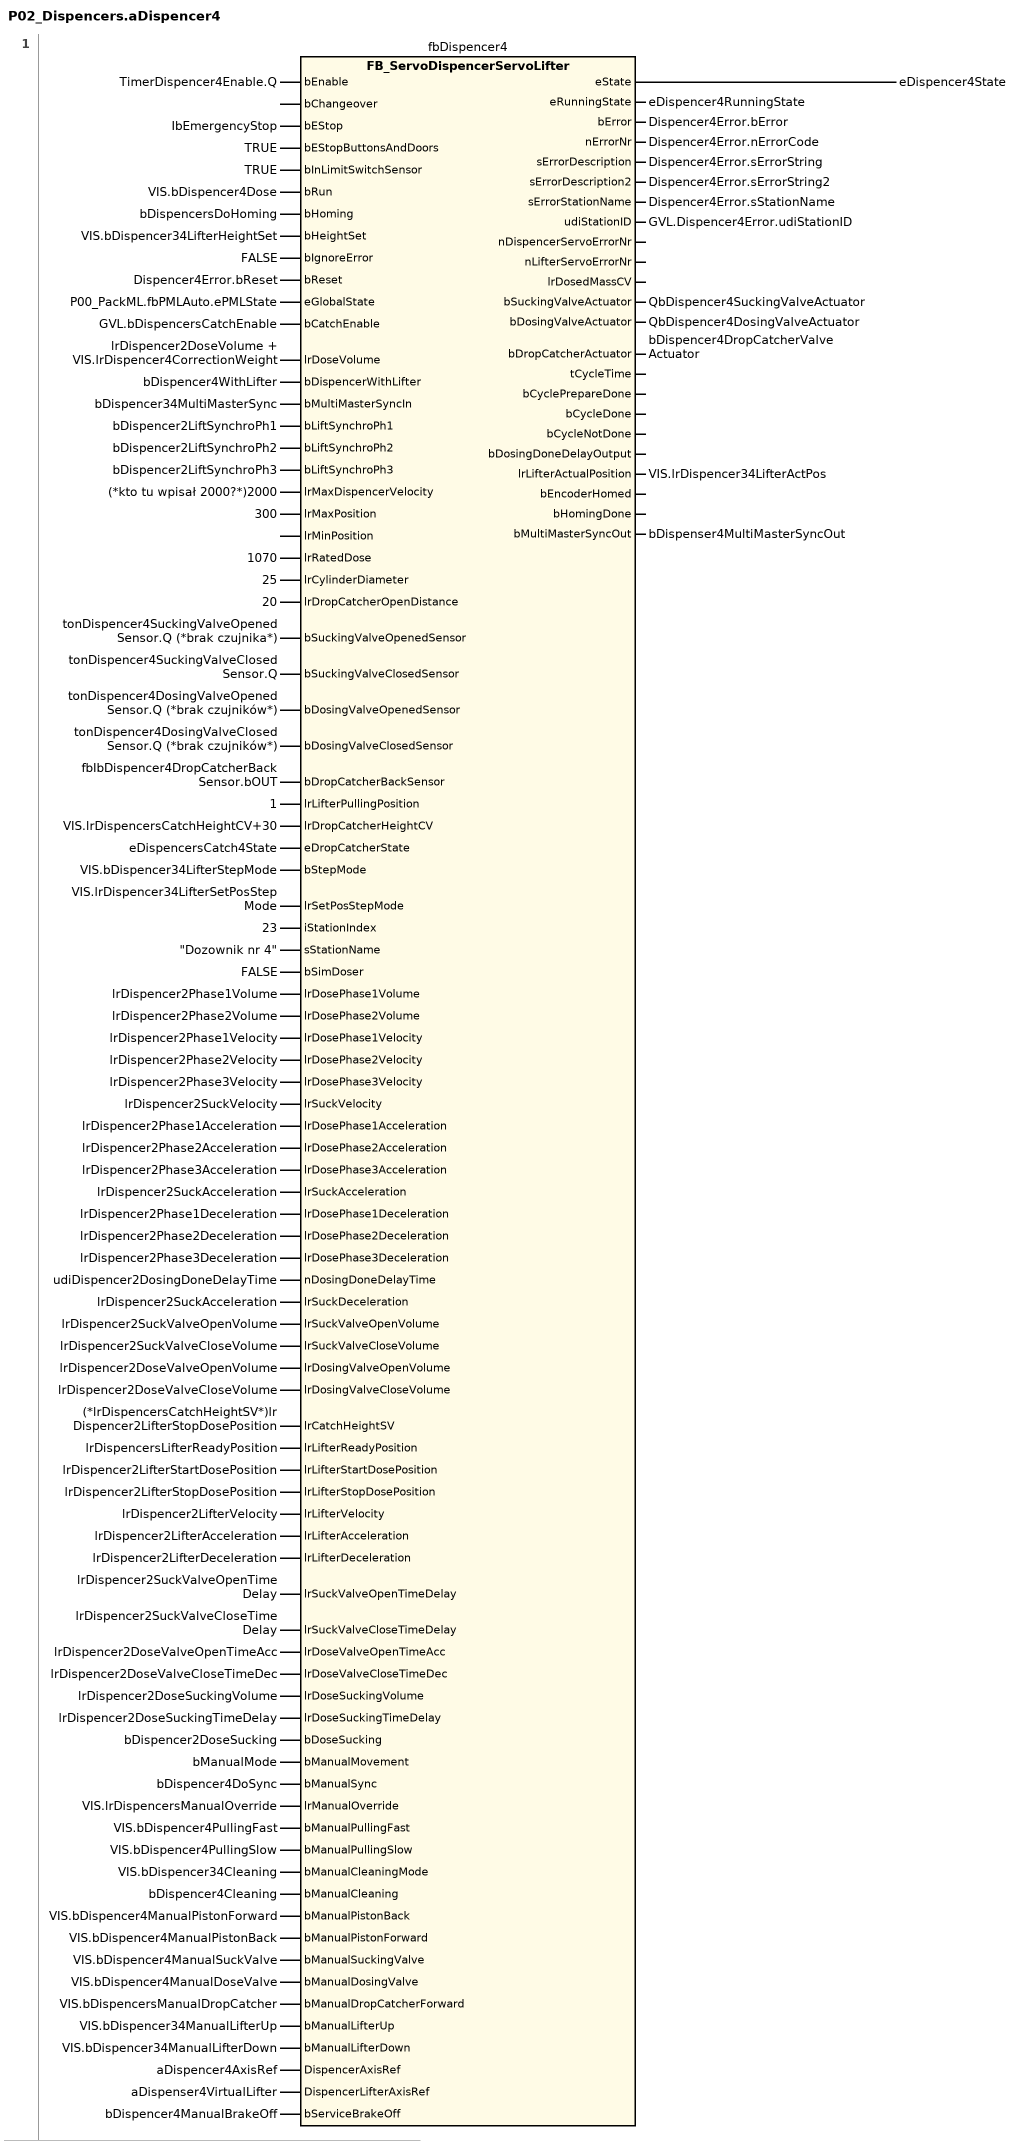
// NETWORK 1
fbDispencer4(
    bEnable := TimerDispencer4Enable.Q,
    bEStop := IbEmergencyStop,
    bEStopButtonsAndDoors := TRUE,
    bInLimitSwitchSensor := TRUE,
    bRun := VIS.bDispencer4Dose,
    bHoming := bDispencersDoHoming,
    bHeightSet := VIS.bDispencer34LifterHeightSet,
    bIgnoreError := FALSE,
    bReset := Dispencer4Error.bReset,
    eGlobalState := P00_PackML.fbPMLAuto.ePMLState,
    bCatchEnable := GVL.bDispencersCatchEnable,
    lrDoseVolume := lrDispencer2DoseVolume + VIS.lrDispencer4CorrectionWeight,
    bDispencerWithLifter := bDispencer4WithLifter,
    bMultiMasterSyncIn := bDispencer34MultiMasterSync,
    bLiftSynchroPh1 := bDispencer2LiftSynchroPh1,
    bLiftSynchroPh2 := bDispencer2LiftSynchroPh2,
    bLiftSynchroPh3 := bDispencer2LiftSynchroPh3,
    lrMaxDispencerVelocity := (*kto tu wpisał 2000?*)2000,
    lrMaxPosition := 300,
    lrRatedDose := 1070,
    lrCylinderDiameter := 25,
    lrDropCatcherOpenDistance := 20,
    bSuckingValveOpenedSensor := tonDispencer4SuckingValveOpenedSensor.Q (*brak czujnika*),
    bSuckingValveClosedSensor := tonDispencer4SuckingValveClosedSensor.Q,
    bDosingValveOpenedSensor := tonDispencer4DosingValveOpenedSensor.Q (*brak czujników*),
    bDosingValveClosedSensor := tonDispencer4DosingValveClosedSensor.Q (*brak czujników*),
    bDropCatcherBackSensor := fbIbDispencer4DropCatcherBackSensor.bOUT,
    lrLifterPullingPosition := 1,
    lrDropCatcherHeightCV := VIS.lrDispencersCatchHeightCV+30,
    eDropCatcherState := eDispencersCatch4State,
    bStepMode := VIS.bDispencer34LifterStepMode,
    lrSetPosStepMode := VIS.lrDispencer34LifterSetPosStepMode,
    iStationIndex := 23,
    sStationName := "Dozownik nr 4",
    bSimDoser := FALSE,
    lrDosePhase1Volume := lrDispencer2Phase1Volume,
    lrDosePhase2Volume := lrDispencer2Phase2Volume,
    lrDosePhase1Velocity := lrDispencer2Phase1Velocity,
    lrDosePhase2Velocity := lrDispencer2Phase2Velocity,
    lrDosePhase3Velocity := lrDispencer2Phase3Velocity,
    lrSuckVelocity := lrDispencer2SuckVelocity,
    lrDosePhase1Acceleration := lrDispencer2Phase1Acceleration,
    lrDosePhase2Acceleration := lrDispencer2Phase2Acceleration,
    lrDosePhase3Acceleration := lrDispencer2Phase3Acceleration,
    lrSuckAcceleration := lrDispencer2SuckAcceleration,
    lrDosePhase1Deceleration := lrDispencer2Phase1Deceleration,
    lrDosePhase2Deceleration := lrDispencer2Phase2Deceleration,
    lrDosePhase3Deceleration := lrDispencer2Phase3Deceleration,
    nDosingDoneDelayTime := udiDispencer2DosingDoneDelayTime,
    lrSuckDeceleration := lrDispencer2SuckAcceleration,
    lrSuckValveOpenVolume := lrDispencer2SuckValveOpenVolume,
    lrSuckValveCloseVolume := lrDispencer2SuckValveCloseVolume,
    lrDosingValveOpenVolume := lrDispencer2DoseValveOpenVolume,
    lrDosingValveCloseVolume := lrDispencer2DoseValveCloseVolume,
    lrCatchHeightSV := (*lrDispencersCatchHeightSV*)lrDispencer2LifterStopDosePosition,
    lrLifterReadyPosition := lrDispencersLifterReadyPosition,
    lrLifterStartDosePosition := lrDispencer2LifterStartDosePosition,
    lrLifterStopDosePosition := lrDispencer2LifterStopDosePosition,
    lrLifterVelocity := lrDispencer2LifterVelocity,
    lrLifterAcceleration := lrDispencer2LifterAcceleration,
    lrLifterDeceleration := lrDispencer2LifterDeceleration,
    lrSuckValveOpenTimeDelay := lrDispencer2SuckValveOpenTimeDelay,
    lrSuckValveCloseTimeDelay := lrDispencer2SuckValveCloseTimeDelay,
    lrDoseValveOpenTimeAcc := lrDispencer2DoseValveOpenTimeAcc,
    lrDoseValveCloseTimeDec := lrDispencer2DoseValveCloseTimeDec,
    lrDoseSuckingVolume := lrDispencer2DoseSuckingVolume,
    lrDoseSuckingTimeDelay := lrDispencer2DoseSuckingTimeDelay,
    bDoseSucking := bDispencer2DoseSucking,
    bManualMovement := bManualMode,
    bManualSync := bDispencer4DoSync,
    lrManualOverride := VIS.lrDispencersManualOverride,
    bManualPullingFast := VIS.bDispencer4PullingFast,
    bManualPullingSlow := VIS.bDispencer4PullingSlow,
    bManualCleaningMode := VIS.bDispencer34Cleaning,
    bManualCleaning := bDispencer4Cleaning,
    bManualPistonBack := VIS.bDispencer4ManualPistonForward,
    bManualPistonForward := VIS.bDispencer4ManualPistonBack,
    bManualSuckingValve := VIS.bDispencer4ManualSuckValve,
    bManualDosingValve := VIS.bDispencer4ManualDoseValve,
    bManualDropCatcherForward := VIS.bDispencersManualDropCatcher,
    bManualLifterUp := VIS.bDispencer34ManualLifterUp,
    bManualLifterDown := VIS.bDispencer34ManualLifterDown,
    DispencerAxisRef := aDispencer4AxisRef,
    DispencerLifterAxisRef := aDispenser4VirtualLifter,
    bServiceBrakeOff := bDispencer4ManualBrakeOff,
    eRunningState => eDispencer4RunningState,
    bError => Dispencer4Error.bError,
    nErrorNr => Dispencer4Error.nErrorCode,
    sErrorDescription => Dispencer4Error.sErrorString,
    sErrorDescription2 => Dispencer4Error.sErrorString2,
    sErrorStationName => Dispencer4Error.sStationName,
    udiStationID => GVL.Dispencer4Error.udiStationID,
    bSuckingValveActuator => QbDispencer4SuckingValveActuator,
    bDosingValveActuator => QbDispencer4DosingValveActuator,
    bDropCatcherActuator => bDispencer4DropCatcherValveActuator,
    lrLifterActualPosition => VIS.lrDispencer34LifterActPos,
    bMultiMasterSyncOut => bDispenser4MultiMasterSyncOut); // FB_ServoDispencerServoLifter
eDispencer4State := fbDispencer4.eState;
END_ACTION

ACTION aDispencerCatch1:
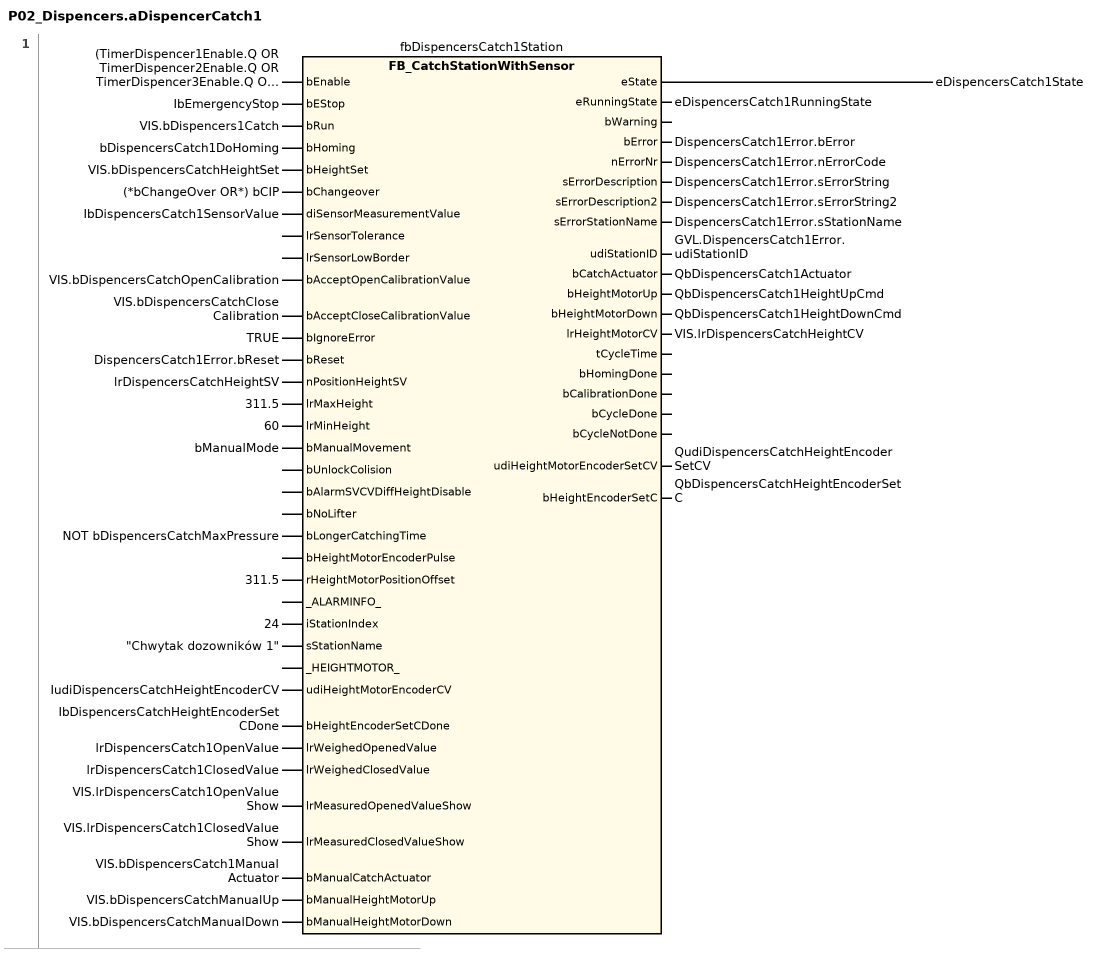
// NETWORK 1
fbDispencersCatch1Station(
    bEnable := (TimerDispencer1Enable.Q OR TimerDispencer2Enable.Q OR TimerDispencer3Enable.Q OR TimerDispencer4Enable.Q)(*AND NOT bChangeOver*) AND NOT bCIP,
    bEStop := IbEmergencyStop,
    bRun := VIS.bDispencers1Catch,
    bHoming := bDispencersCatch1DoHoming,
    bHeightSet := VIS.bDispencersCatchHeightSet,
    bChangeover := (*bChangeOver OR*) bCIP,
    diSensorMeasurementValue := IbDispencersCatch1SensorValue,
    bAcceptOpenCalibrationValue := VIS.bDispencersCatchOpenCalibration,
    bAcceptCloseCalibrationValue := VIS.bDispencersCatchCloseCalibration,
    bIgnoreError := TRUE,
    bReset := DispencersCatch1Error.bReset,
    nPositionHeightSV := lrDispencersCatchHeightSV,
    lrMaxHeight := 311.5,
    lrMinHeight := 60,
    bManualMovement := bManualMode,
    bLongerCatchingTime := NOT bDispencersCatchMaxPressure,
    rHeightMotorPositionOffset := 311.5,
    iStationIndex := 24,
    sStationName := "Chwytak dozowników 1",
    udiHeightMotorEncoderCV := IudiDispencersCatchHeightEncoderCV,
    bHeightEncoderSetCDone := IbDispencersCatchHeightEncoderSetCDone,
    lrWeighedOpenedValue := lrDispencersCatch1OpenValue,
    lrWeighedClosedValue := lrDispencersCatch1ClosedValue,
    lrMeasuredOpenedValueShow := VIS.lrDispencersCatch1OpenValueShow,
    lrMeasuredClosedValueShow := VIS.lrDispencersCatch1ClosedValueShow,
    bManualCatchActuator := VIS.bDispencersCatch1ManualActuator,
    bManualHeightMotorUp := VIS.bDispencersCatchManualUp,
    bManualHeightMotorDown := VIS.bDispencersCatchManualDown,
    eRunningState => eDispencersCatch1RunningState,
    bError => DispencersCatch1Error.bError,
    nErrorNr => DispencersCatch1Error.nErrorCode,
    sErrorDescription => DispencersCatch1Error.sErrorString,
    sErrorDescription2 => DispencersCatch1Error.sErrorString2,
    sErrorStationName => DispencersCatch1Error.sStationName,
    udiStationID => GVL.DispencersCatch1Error.udiStationID,
    bCatchActuator => QbDispencersCatch1Actuator,
    bHeightMotorUp => QbDispencersCatch1HeightUpCmd,
    bHeightMotorDown => QbDispencersCatch1HeightDownCmd,
    lrHeightMotorCV => VIS.lrDispencersCatchHeightCV,
    udiHeightMotorEncoderSetCV => QudiDispencersCatchHeightEncoderSetCV,
    bHeightEncoderSetC => QbDispencersCatchHeightEncoderSetC); // FB_CatchStationWithSensor
eDispencersCatch1State := fbDispencersCatch1Station.eState;
END_ACTION

ACTION aDispencerCatch2:
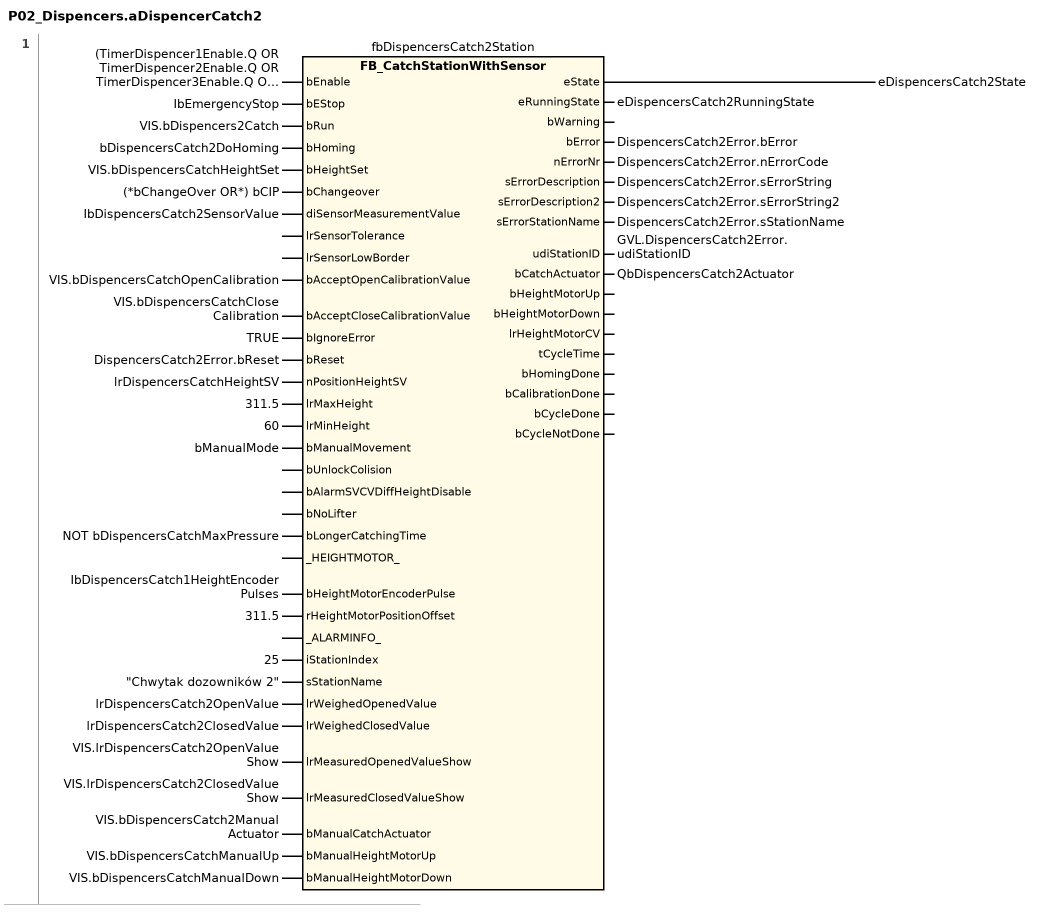
// NETWORK 1
fbDispencersCatch2Station(
    bEnable := (TimerDispencer1Enable.Q OR TimerDispencer2Enable.Q OR TimerDispencer3Enable.Q OR TimerDispencer4Enable.Q)(*AND NOT bChangeOver*) AND NOT bCIP,
    bEStop := IbEmergencyStop,
    bRun := VIS.bDispencers2Catch,
    bHoming := bDispencersCatch2DoHoming,
    bHeightSet := VIS.bDispencersCatchHeightSet,
    bChangeover := (*bChangeOver OR*) bCIP,
    diSensorMeasurementValue := IbDispencersCatch2SensorValue,
    bAcceptOpenCalibrationValue := VIS.bDispencersCatchOpenCalibration,
    bAcceptCloseCalibrationValue := VIS.bDispencersCatchCloseCalibration,
    bIgnoreError := TRUE,
    bReset := DispencersCatch2Error.bReset,
    nPositionHeightSV := lrDispencersCatchHeightSV,
    lrMaxHeight := 311.5,
    lrMinHeight := 60,
    bManualMovement := bManualMode,
    bLongerCatchingTime := NOT bDispencersCatchMaxPressure,
    bHeightMotorEncoderPulse := IbDispencersCatch1HeightEncoderPulses,
    rHeightMotorPositionOffset := 311.5,
    iStationIndex := 25,
    sStationName := "Chwytak dozowników 2",
    lrWeighedOpenedValue := lrDispencersCatch2OpenValue,
    lrWeighedClosedValue := lrDispencersCatch2ClosedValue,
    lrMeasuredOpenedValueShow := VIS.lrDispencersCatch2OpenValueShow,
    lrMeasuredClosedValueShow := VIS.lrDispencersCatch2ClosedValueShow,
    bManualCatchActuator := VIS.bDispencersCatch2ManualActuator,
    bManualHeightMotorUp := VIS.bDispencersCatchManualUp,
    bManualHeightMotorDown := VIS.bDispencersCatchManualDown,
    eRunningState => eDispencersCatch2RunningState,
    bError => DispencersCatch2Error.bError,
    nErrorNr => DispencersCatch2Error.nErrorCode,
    sErrorDescription => DispencersCatch2Error.sErrorString,
    sErrorDescription2 => DispencersCatch2Error.sErrorString2,
    sErrorStationName => DispencersCatch2Error.sStationName,
    udiStationID => GVL.DispencersCatch2Error.udiStationID,
    bCatchActuator => QbDispencersCatch2Actuator); // FB_CatchStationWithSensor
eDispencersCatch2State := fbDispencersCatch2Station.eState;
END_ACTION

ACTION aDispencerCatch3:
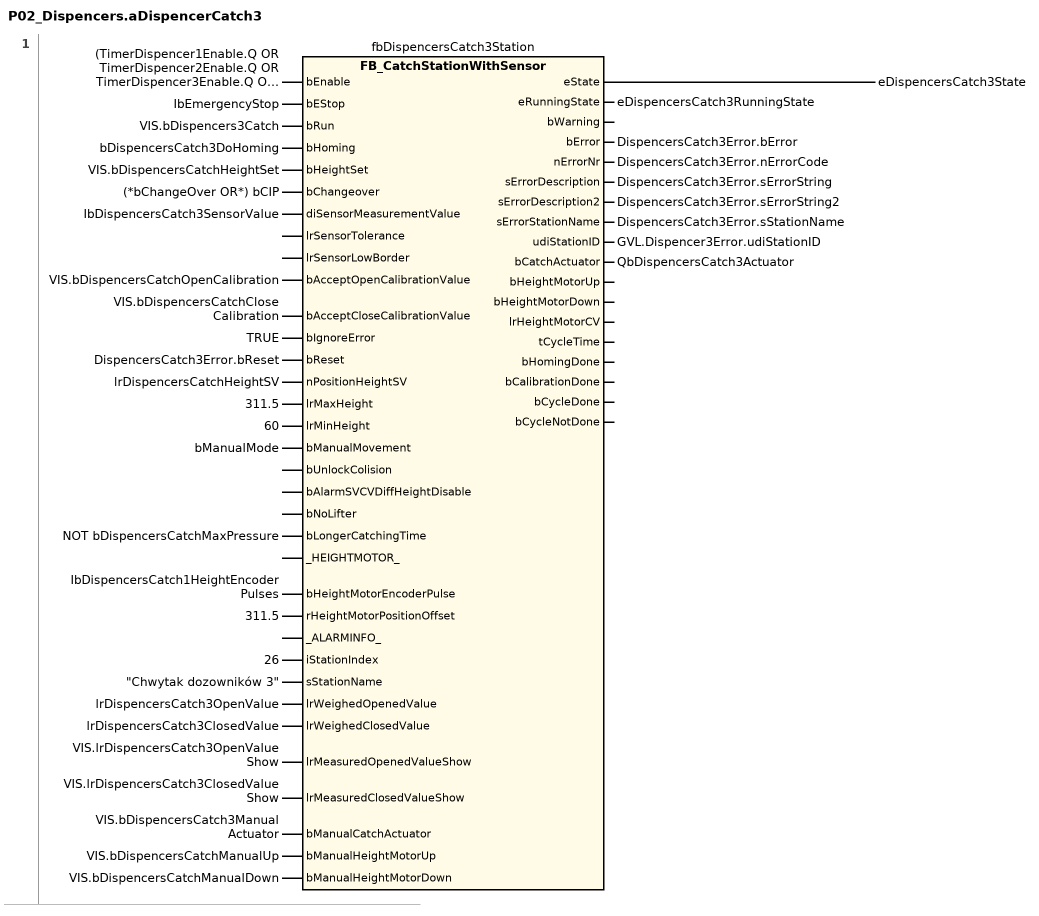
// NETWORK 1
fbDispencersCatch3Station(
    bEnable := (TimerDispencer1Enable.Q OR TimerDispencer2Enable.Q OR TimerDispencer3Enable.Q OR TimerDispencer4Enable.Q) (*AND NOT bChangeOver*) AND NOT bCIP,
    bEStop := IbEmergencyStop,
    bRun := VIS.bDispencers3Catch,
    bHoming := bDispencersCatch3DoHoming,
    bHeightSet := VIS.bDispencersCatchHeightSet,
    bChangeover := (*bChangeOver OR*) bCIP,
    diSensorMeasurementValue := IbDispencersCatch3SensorValue,
    bAcceptOpenCalibrationValue := VIS.bDispencersCatchOpenCalibration,
    bAcceptCloseCalibrationValue := VIS.bDispencersCatchCloseCalibration,
    bIgnoreError := TRUE,
    bReset := DispencersCatch3Error.bReset,
    nPositionHeightSV := lrDispencersCatchHeightSV,
    lrMaxHeight := 311.5,
    lrMinHeight := 60,
    bManualMovement := bManualMode,
    bLongerCatchingTime := NOT bDispencersCatchMaxPressure,
    bHeightMotorEncoderPulse := IbDispencersCatch1HeightEncoderPulses,
    rHeightMotorPositionOffset := 311.5,
    iStationIndex := 26,
    sStationName := "Chwytak dozowników 3",
    lrWeighedOpenedValue := lrDispencersCatch3OpenValue,
    lrWeighedClosedValue := lrDispencersCatch3ClosedValue,
    lrMeasuredOpenedValueShow := VIS.lrDispencersCatch3OpenValueShow,
    lrMeasuredClosedValueShow := VIS.lrDispencersCatch3ClosedValueShow,
    bManualCatchActuator := VIS.bDispencersCatch3ManualActuator,
    bManualHeightMotorUp := VIS.bDispencersCatchManualUp,
    bManualHeightMotorDown := VIS.bDispencersCatchManualDown,
    eRunningState => eDispencersCatch3RunningState,
    bError => DispencersCatch3Error.bError,
    nErrorNr => DispencersCatch3Error.nErrorCode,
    sErrorDescription => DispencersCatch3Error.sErrorString,
    sErrorDescription2 => DispencersCatch3Error.sErrorString2,
    sErrorStationName => DispencersCatch3Error.sStationName,
    udiStationID => GVL.Dispencer3Error.udiStationID,
    bCatchActuator => QbDispencersCatch3Actuator); // FB_CatchStationWithSensor
eDispencersCatch3State := fbDispencersCatch3Station.eState;
END_ACTION

ACTION aDispencerCatch4:
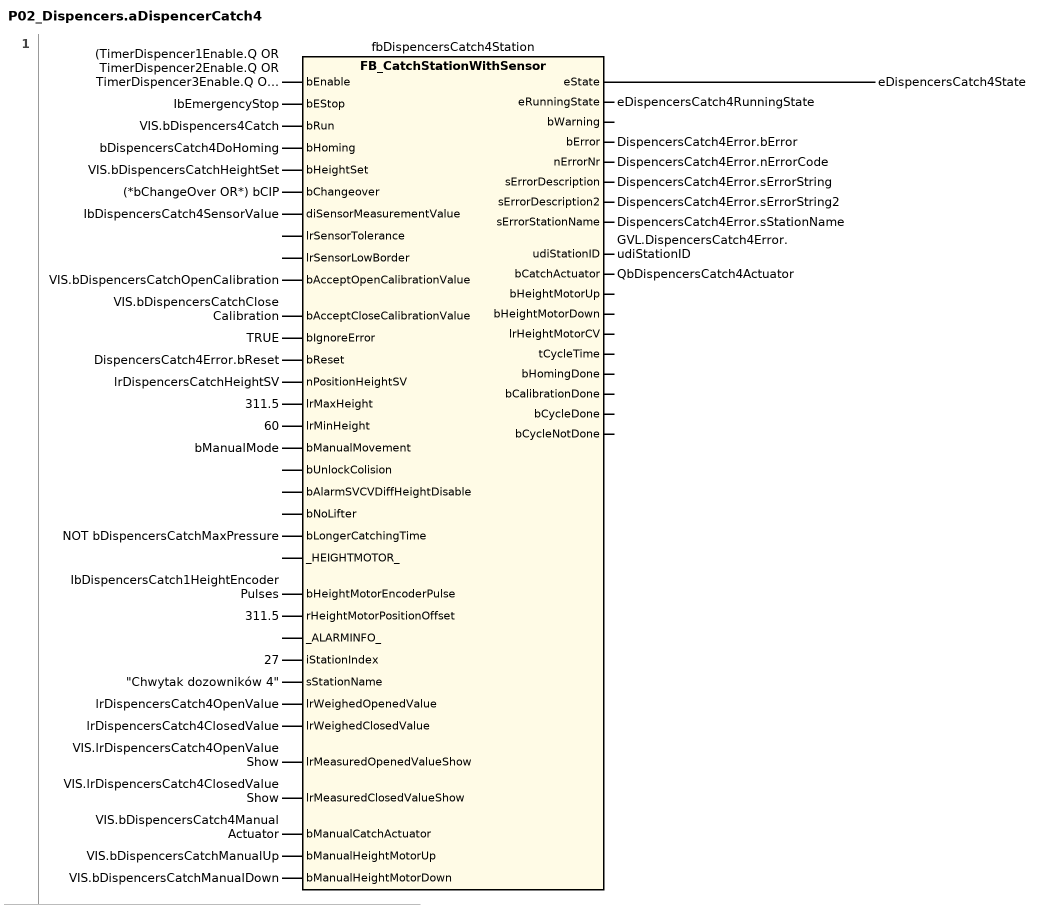
// NETWORK 1
fbDispencersCatch4Station(
    bEnable := (TimerDispencer1Enable.Q OR TimerDispencer2Enable.Q OR TimerDispencer3Enable.Q OR TimerDispencer4Enable.Q) (*AND NOT bChangeOver*) AND NOT bCIP,
    bEStop := IbEmergencyStop,
    bRun := VIS.bDispencers4Catch,
    bHoming := bDispencersCatch4DoHoming,
    bHeightSet := VIS.bDispencersCatchHeightSet,
    bChangeover := (*bChangeOver OR*) bCIP,
    diSensorMeasurementValue := IbDispencersCatch4SensorValue,
    bAcceptOpenCalibrationValue := VIS.bDispencersCatchOpenCalibration,
    bAcceptCloseCalibrationValue := VIS.bDispencersCatchCloseCalibration,
    bIgnoreError := TRUE,
    bReset := DispencersCatch4Error.bReset,
    nPositionHeightSV := lrDispencersCatchHeightSV,
    lrMaxHeight := 311.5,
    lrMinHeight := 60,
    bManualMovement := bManualMode,
    bLongerCatchingTime := NOT bDispencersCatchMaxPressure,
    bHeightMotorEncoderPulse := IbDispencersCatch1HeightEncoderPulses,
    rHeightMotorPositionOffset := 311.5,
    iStationIndex := 27,
    sStationName := "Chwytak dozowników 4",
    lrWeighedOpenedValue := lrDispencersCatch4OpenValue,
    lrWeighedClosedValue := lrDispencersCatch4ClosedValue,
    lrMeasuredOpenedValueShow := VIS.lrDispencersCatch4OpenValueShow,
    lrMeasuredClosedValueShow := VIS.lrDispencersCatch4ClosedValueShow,
    bManualCatchActuator := VIS.bDispencersCatch4ManualActuator,
    bManualHeightMotorUp := VIS.bDispencersCatchManualUp,
    bManualHeightMotorDown := VIS.bDispencersCatchManualDown,
    eRunningState => eDispencersCatch4RunningState,
    bError => DispencersCatch4Error.bError,
    nErrorNr => DispencersCatch4Error.nErrorCode,
    sErrorDescription => DispencersCatch4Error.sErrorString,
    sErrorDescription2 => DispencersCatch4Error.sErrorString2,
    sErrorStationName => DispencersCatch4Error.sStationName,
    udiStationID => GVL.DispencersCatch4Error.udiStationID,
    bCatchActuator => QbDispencersCatch4Actuator); // FB_CatchStationWithSensor
eDispencersCatch4State := fbDispencersCatch4Station.eState;
END_ACTION

ACTION aDispencerCatchPressure:


P02_Dispencers.QbDispencersCatchMaxPressure := bDispencersCatchMaxPressure;
END_ACTION

ACTION aDispencerDragStation:
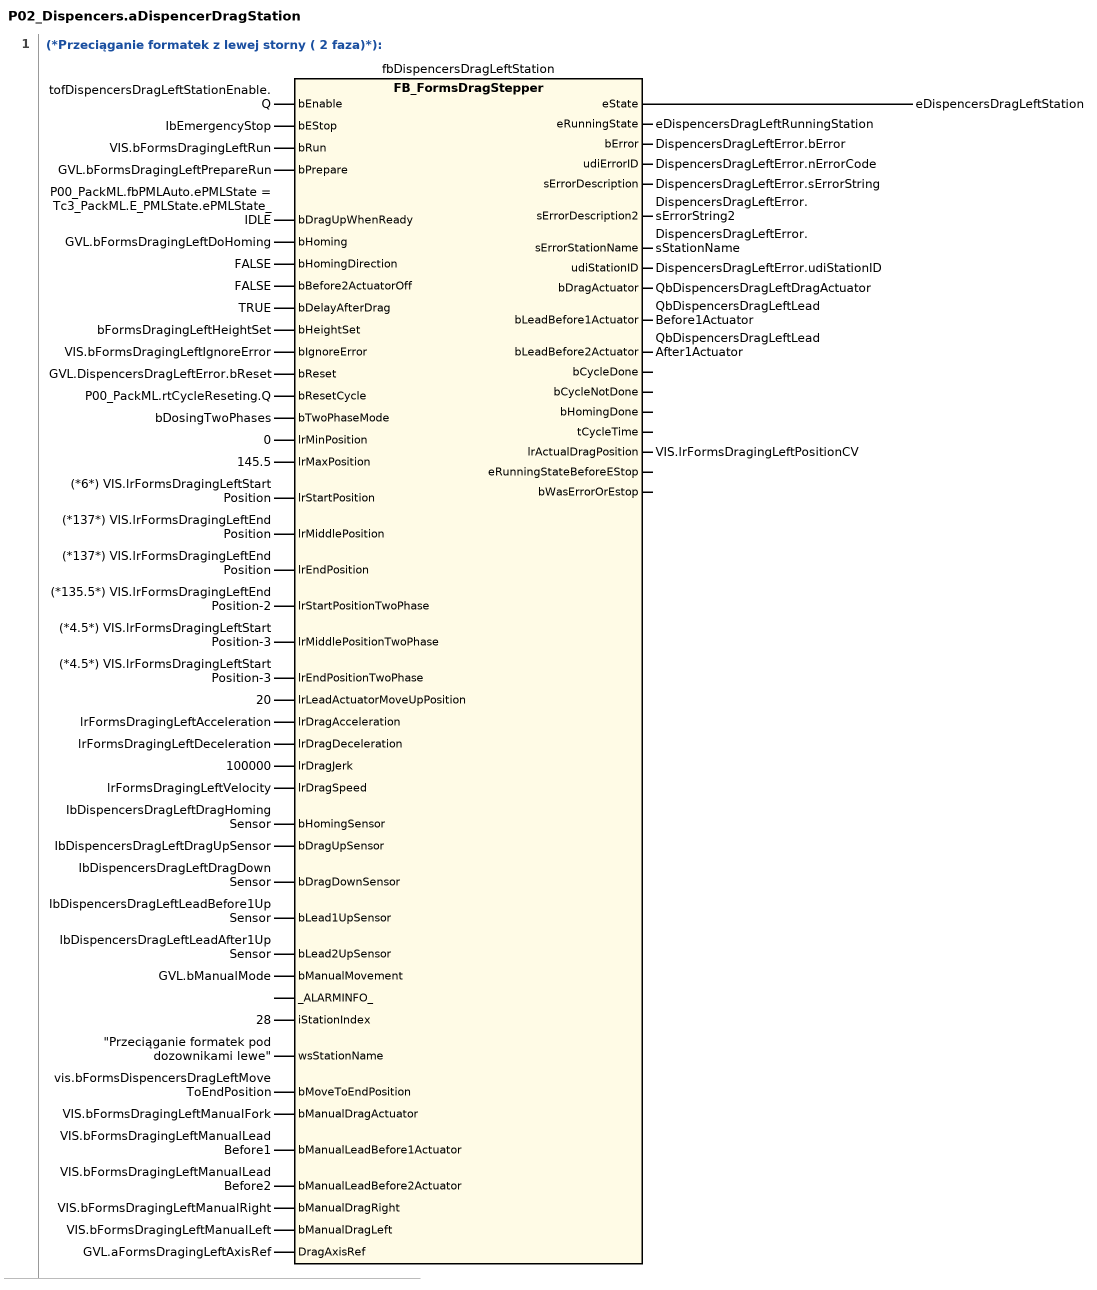
// NETWORK 1
// label: (*Przeciąganie formatek z lewej storny ( 2 faza)*)
fbDispencersDragLeftStation(
    bEnable := tofDispencersDragLeftStationEnable.Q,
    bEStop := IbEmergencyStop,
    bRun := VIS.bFormsDragingLeftRun,
    bPrepare := GVL.bFormsDragingLeftPrepareRun,
    bDragUpWhenReady := P00_PackML.fbPMLAuto.ePMLState = Tc3_PackML.E_PMLState.ePMLState_IDLE,
    bHoming := GVL.bFormsDragingLeftDoHoming,
    bHomingDirection := FALSE,
    bBefore2ActuatorOff := FALSE,
    bDelayAfterDrag := TRUE,
    bHeightSet := bFormsDragingLeftHeightSet,
    bIgnoreError := VIS.bFormsDragingLeftIgnoreError,
    bReset := GVL.DispencersDragLeftError.bReset,
    bResetCycle := P00_PackML.rtCycleReseting.Q,
    bTwoPhaseMode := bDosingTwoPhases,
    lrMinPosition := 0,
    lrMaxPosition := 145.5,
    lrStartPosition := (*6*) VIS.lrFormsDragingLeftStartPosition,
    lrMiddlePosition := (*137*) VIS.lrFormsDragingLeftEndPosition,
    lrEndPosition := (*137*) VIS.lrFormsDragingLeftEndPosition,
    lrStartPositionTwoPhase := (*135.5*) VIS.lrFormsDragingLeftEndPosition-2,
    lrMiddlePositionTwoPhase := (*4.5*) VIS.lrFormsDragingLeftStartPosition-3,
    lrEndPositionTwoPhase := (*4.5*) VIS.lrFormsDragingLeftStartPosition-3,
    lrLeadActuatorMoveUpPosition := 20,
    lrDragAcceleration := lrFormsDragingLeftAcceleration,
    lrDragDeceleration := lrFormsDragingLeftDeceleration,
    lrDragJerk := 100000,
    lrDragSpeed := lrFormsDragingLeftVelocity,
    bHomingSensor := IbDispencersDragLeftDragHomingSensor,
    bDragUpSensor := IbDispencersDragLeftDragUpSensor,
    bDragDownSensor := IbDispencersDragLeftDragDownSensor,
    bLead1UpSensor := IbDispencersDragLeftLeadBefore1UpSensor,
    bLead2UpSensor := IbDispencersDragLeftLeadAfter1UpSensor,
    bManualMovement := GVL.bManualMode,
    iStationIndex := 28,
    wsStationName := "Przeciąganie formatek pod dozownikami lewe",
    bMoveToEndPosition := vis.bFormsDispencersDragLeftMoveToEndPosition,
    bManualDragActuator := VIS.bFormsDragingLeftManualFork,
    bManualLeadBefore1Actuator := VIS.bFormsDragingLeftManualLeadBefore1,
    bManualLeadBefore2Actuator := VIS.bFormsDragingLeftManualLeadBefore2,
    bManualDragRight := VIS.bFormsDragingLeftManualRight,
    bManualDragLeft := VIS.bFormsDragingLeftManualLeft,
    DragAxisRef := GVL.aFormsDragingLeftAxisRef,
    eRunningState => eDispencersDragLeftRunningStation,
    bError => DispencersDragLeftError.bError,
    udiErrorID => DispencersDragLeftError.nErrorCode,
    sErrorDescription => DispencersDragLeftError.sErrorString,
    sErrorDescription2 => DispencersDragLeftError.sErrorString2,
    sErrorStationName => DispencersDragLeftError.sStationName,
    udiStationID => DispencersDragLeftError.udiStationID,
    bDragActuator => QbDispencersDragLeftDragActuator,
    bLeadBefore1Actuator => QbDispencersDragLeftLeadBefore1Actuator,
    bLeadBefore2Actuator => QbDispencersDragLeftLeadAfter1Actuator,
    lrActualDragPosition => VIS.lrFormsDragingLeftPositionCV); // FB_FormsDragStepper
eDispencersDragLeftStation := fbDispencersDragLeftStation.eState;

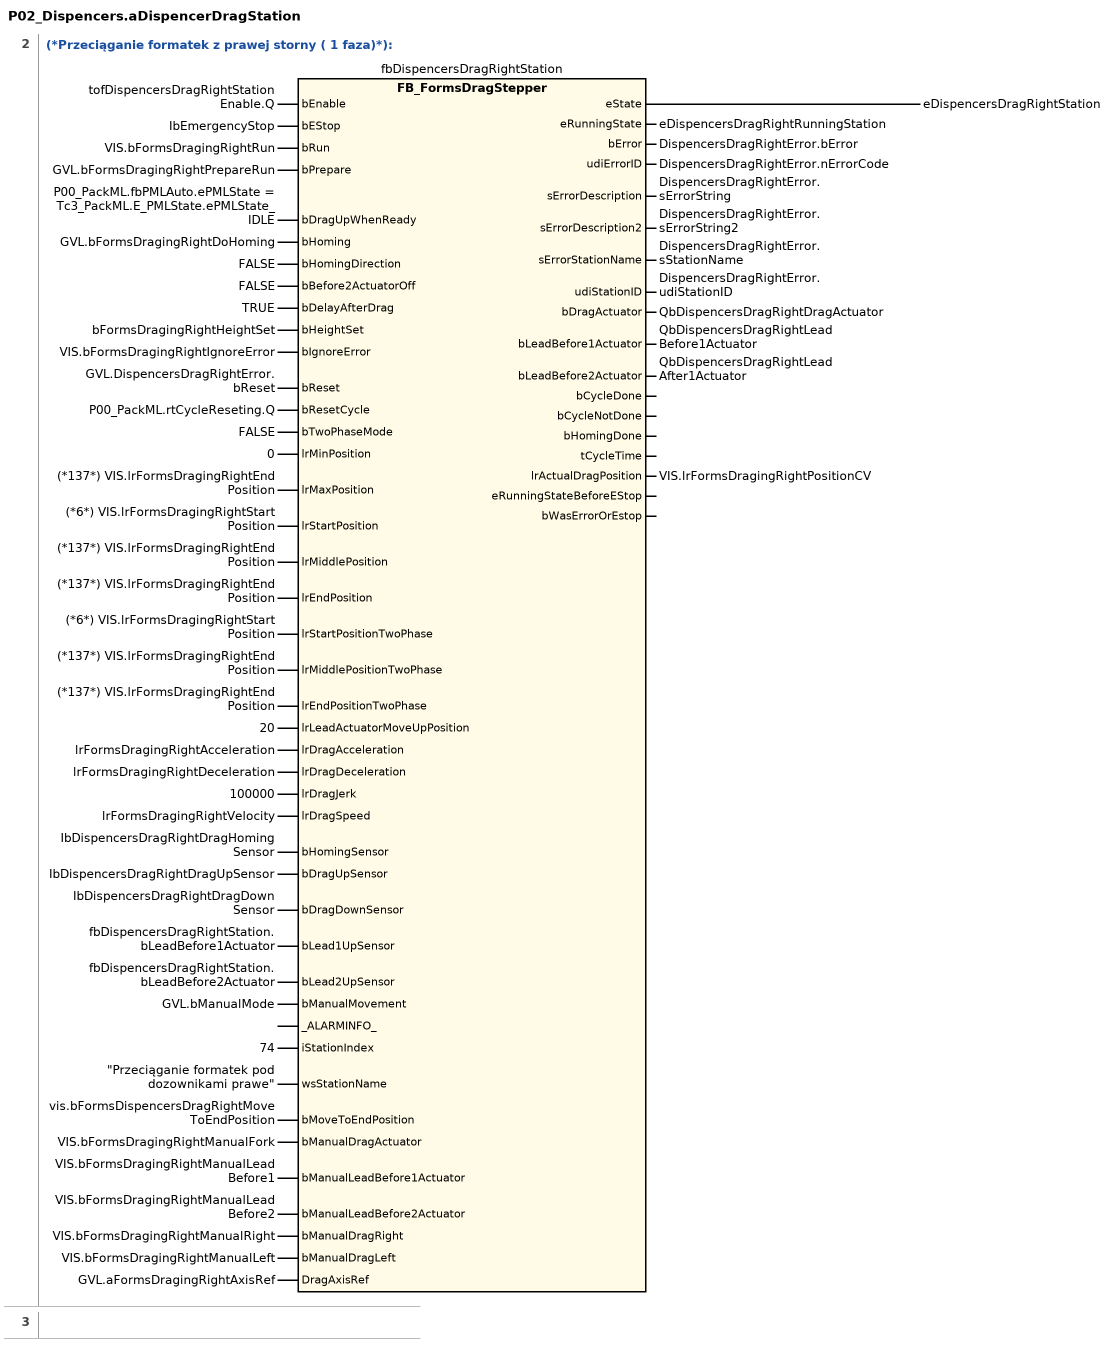
// NETWORK 2
// label: (*Przeciąganie formatek z prawej storny ( 1 faza)*)
fbDispencersDragRightStation(
    bEnable := tofDispencersDragRightStationEnable.Q,
    bEStop := IbEmergencyStop,
    bRun := VIS.bFormsDragingRightRun,
    bPrepare := GVL.bFormsDragingRightPrepareRun,
    bDragUpWhenReady := P00_PackML.fbPMLAuto.ePMLState = Tc3_PackML.E_PMLState.ePMLState_IDLE,
    bHoming := GVL.bFormsDragingRightDoHoming,
    bHomingDirection := FALSE,
    bBefore2ActuatorOff := FALSE,
    bDelayAfterDrag := TRUE,
    bHeightSet := bFormsDragingRightHeightSet,
    bIgnoreError := VIS.bFormsDragingRightIgnoreError,
    bReset := GVL.DispencersDragRightError.bReset,
    bResetCycle := P00_PackML.rtCycleReseting.Q,
    bTwoPhaseMode := FALSE,
    lrMinPosition := 0,
    lrMaxPosition := (*137*) VIS.lrFormsDragingRightEndPosition,
    lrStartPosition := (*6*) VIS.lrFormsDragingRightStartPosition,
    lrMiddlePosition := (*137*) VIS.lrFormsDragingRightEndPosition,
    lrEndPosition := (*137*) VIS.lrFormsDragingRightEndPosition,
    lrStartPositionTwoPhase := (*6*) VIS.lrFormsDragingRightStartPosition,
    lrMiddlePositionTwoPhase := (*137*) VIS.lrFormsDragingRightEndPosition,
    lrEndPositionTwoPhase := (*137*) VIS.lrFormsDragingRightEndPosition,
    lrLeadActuatorMoveUpPosition := 20,
    lrDragAcceleration := lrFormsDragingRightAcceleration,
    lrDragDeceleration := lrFormsDragingRightDeceleration,
    lrDragJerk := 100000,
    lrDragSpeed := lrFormsDragingRightVelocity,
    bHomingSensor := IbDispencersDragRightDragHomingSensor,
    bDragUpSensor := IbDispencersDragRightDragUpSensor,
    bDragDownSensor := IbDispencersDragRightDragDownSensor,
    bLead1UpSensor := fbDispencersDragRightStation.bLeadBefore1Actuator,
    bLead2UpSensor := fbDispencersDragRightStation.bLeadBefore2Actuator,
    bManualMovement := GVL.bManualMode,
    iStationIndex := 74,
    wsStationName := "Przeciąganie formatek pod dozownikami prawe",
    bMoveToEndPosition := vis.bFormsDispencersDragRightMoveToEndPosition,
    bManualDragActuator := VIS.bFormsDragingRightManualFork,
    bManualLeadBefore1Actuator := VIS.bFormsDragingRightManualLeadBefore1,
    bManualLeadBefore2Actuator := VIS.bFormsDragingRightManualLeadBefore2,
    bManualDragRight := VIS.bFormsDragingRightManualRight,
    bManualDragLeft := VIS.bFormsDragingRightManualLeft,
    DragAxisRef := GVL.aFormsDragingRightAxisRef,
    eRunningState => eDispencersDragRightRunningStation,
    bError => DispencersDragRightError.bError,
    udiErrorID => DispencersDragRightError.nErrorCode,
    sErrorDescription => DispencersDragRightError.sErrorString,
    sErrorDescription2 => DispencersDragRightError.sErrorString2,
    sErrorStationName => DispencersDragRightError.sStationName,
    udiStationID => DispencersDragRightError.udiStationID,
    bDragActuator => QbDispencersDragRightDragActuator,
    bLeadBefore1Actuator => QbDispencersDragRightLeadBefore1Actuator,
    bLeadBefore2Actuator => QbDispencersDragRightLeadAfter1Actuator,
    lrActualDragPosition => VIS.lrFormsDragingRightPositionCV); // FB_FormsDragStepper
eDispencersDragRightStation := fbDispencersDragRightStation.eState;

// NETWORK 3
END_ACTION

ACTION aDispencersCatchWarnings:
tonDispencersWarningReset(IN:=DispencersWarning[0].bWarning OR DispencersWarning[1].bWarning OR DispencersWarning[2].bWarning OR DispencersWarning[3].bWarning
						,PT:=T#10S);
						
IF tonDispencersWarningReset.Q THEN
	DispencersWarning[0].bAcknowledge := TRUE;
	DispencersWarning[1].bAcknowledge := TRUE;
	DispencersWarning[2].bAcknowledge := TRUE;
	DispencersWarning[3].bAcknowledge := TRUE;
END_IF

//Nieskalibrowany czujnika chwytaka 1 2 3 4

IF fbDispencersCatch1Station.bWarning OR fbDispencersCatch2Station.bWarning OR fbDispencersCatch3Station.bWarning OR fbDispencersCatch4Station.bWarning 
	AND fbDispencersCatch1Station.bEnable AND NOT DispencersWarning[0].bWarning THEN
	DispencersWarning[0].bWarning												:=TRUE;
	DispencersWarning[0].udiWarningCode											:=17;
	DispencersWarning[0].sDescription											:='Dozowniki | Nieskalibrowany czujnik chwytaka szyjek pod dozownikami';
ELSIF NOT fbDispencersCatch1Station.bWarning AND NOT fbDispencersCatch2Station.bWarning AND NOT fbDispencersCatch3Station.bWarning AND NOT fbDispencersCatch4Station.bWarning  AND DispencersWarning[0].bAcknowledge THEN
	DispencersWarning[0].bWarning												:=FALSE;
	DispencersWarning[0].bAcknowledge											:=FALSE;
	VIS.uliWarningAcknowledge.10 												:=FALSE;
ELSIF DispencersWarning[0].bAcknowledge THEN
	DispencersWarning[0].bAcknowledge											:=TRUE;
END_IF

//Niechwycona butelka chwytaka dozownika 1
IF fbDispencersCatch1Station.eRunningState = E_CatchStationState.eNotCatched AND NOT DispencersWarning[1].bWarning THEN
	DispencersWarning[1].bWarning												:=TRUE;
	DispencersWarning[1].udiWarningCode											:=18;
	DispencersWarning[1].sDescription											:='Dozowniki | Nieprawidłowo chwycona butelka przez chwytak dozownika 1';
ELSIF fbDispencersCatch1Station.eRunningState <> E_CatchStationState.eNotCatched AND DispencersWarning[1].bAcknowledge THEN
	DispencersWarning[1].bWarning												:=FALSE;
	DispencersWarning[1].bAcknowledge											:=FALSE;
	VIS.uliWarningAcknowledge.11 												:=FALSE;
ELSIF DispencersWarning[1].bAcknowledge THEN
	DispencersWarning[1].bAcknowledge											:=TRUE;
END_IF

//Niechwycona butelka chwytaka dozownika 2
IF fbDispencersCatch2Station.eRunningState = E_CatchStationState.eNotCatched AND NOT DispencersWarning[2].bWarning THEN
	DispencersWarning[2].bWarning												:=TRUE;
	DispencersWarning[2].udiWarningCode											:=19;
	DispencersWarning[2].sDescription											:='Dozowniki | Nieprawidłowo chwycona butelka przez chwytak dozownika 2';
ELSIF fbDispencersCatch2Station.eRunningState <> E_CatchStationState.eNotCatched AND DispencersWarning[2].bAcknowledge THEN
	DispencersWarning[2].bWarning												:=FALSE;
	DispencersWarning[2].bAcknowledge											:=FALSE;
	VIS.uliWarningAcknowledge.12 												:=FALSE;
ELSIF DispencersWarning[2].bAcknowledge THEN
	DispencersWarning[2].bAcknowledge											:=TRUE;
END_IF

//Niechwycona butelka chwytaka dozownika 3
IF fbDispencersCatch3Station.eRunningState = E_CatchStationState.eNotCatched AND NOT DispencersWarning[3].bWarning THEN
	DispencersWarning[3].bWarning												:=TRUE;
	DispencersWarning[3].udiWarningCode											:=20;
	DispencersWarning[3].sDescription											:='Dozowniki | Nieprawidłowo chwycona butelka przez chwytak dozownika 3';
ELSIF fbDispencersCatch2Station.eRunningState <> E_CatchStationState.eNotCatched AND DispencersWarning[3].bAcknowledge THEN
	DispencersWarning[3].bWarning												:=FALSE;
	DispencersWarning[3].bAcknowledge											:=FALSE;
	VIS.uliWarningAcknowledge.13 												:=FALSE;
ELSIF DispencersWarning[3].bAcknowledge THEN
	DispencersWarning[3].bAcknowledge											:=TRUE;
END_IF

//Niechwycona butelka chwytaka dozownika 4
IF fbDispencersCatch4Station.eRunningState = E_CatchStationState.eNotCatched AND NOT DispencersWarning[4].bWarning THEN
	DispencersWarning[4].bWarning:=TRUE;
	DispencersWarning[4].udiWarningCode											:=21;
	DispencersWarning[4].sDescription											:='Dozowniki | Nieprawidłowo chwycona butelka przez chwytak dozownika 4';
ELSIF fbDispencersCatch2Station.eRunningState <> E_CatchStationState.eNotCatched AND DispencersWarning[4].bAcknowledge THEN
	DispencersWarning[4].bWarning		:=	FALSE;
	DispencersWarning[4].bAcknowledge	:=	FALSE;
	VIS.uliWarningAcknowledge.14 := FALSE;
ELSIF DispencersWarning[4].bAcknowledge THEN
	DispencersWarning[4].bAcknowledge	:=	TRUE;
END_IF
END_ACTION

ACTION aDispencersDragStationLeadActuators:

//QbDispencersDragLeftLeadBefore1Actuator := fbDispencersDragLeftStation.bLeadBefore1Actuator AND fbDispencersDragRightStation.bLeadBefore1Actuator;
//QbDispencersDragLeftLeadAfter1Actuator	:= fbDispencersDragLeftStation.bLeadBefore2Actuator AND fbDispencersDragRightStation.bLeadBefore2Actuator;
END_ACTION

ACTION aDispencersEnable:
(*Opoznienie wyłączanie enabla dozownikow*)
(*Nie zdarzy wyjśc z Disabled podczas zmiany recepptury*)
TimerDispencer1Enable			(IN := bDispencer1Enable, PT := T#3S);
TimerDispencer2Enable			(IN := bDispencer2Enable, PT := T#3S);
TimerDispencer3Enable			(IN := bDispencer3Enable, PT := T#3S);
TimerDispencer4Enable			(IN := bDispencer4Enable, PT := T#3S);

(*Wyłączanie dozowników parami*)
//bDispencer1Enable				:= bDispencer1Enable AND bDispencer2Enable AND bDispencer3Enable AND bDispencer4Enable;
//bDispencer2Enable 			:= bDispencer1Enable AND bDispencer2Enable AND bDispencer3Enable AND bDispencer4Enable;
bDispencer1Enable				:= bDispencer1Enable AND bDispencer2Enable;
bDispencer2Enable 				:= bDispencer1Enable AND bDispencer2Enable;
bDispencer3Enable				:= bDispencer3Enable AND bDispencer4Enable;
bDispencer4Enable 				:= bDispencer3Enable AND bDispencer4Enable;

(*Ustawianie zmiennych wizualizacyjnych*)
rtbDispencer12EnableShow		(CLK:=VIS.bDispencer1EnableShow OR VIS.bDispencer2EnableShow,Q=>);
IF rtbDispencer12EnableShow.Q THEN
	VIS.bDispencer1EnableShow 	:= TRUE;
	VIS.bDispencer2EnableShow 	:= TRUE;	
END_IF
ftbDispencer12EnableShow		(CLK:=VIS.bDispencer1EnableShow AND VIS.bDispencer2EnableShow,Q=>);
IF ftbDispencer12EnableShow.Q THEN
	VIS.bDispencer1EnableShow 	:= FALSE;
	VIS.bDispencer2EnableShow 	:= FALSE;	
END_IF


(*Ustawianie zmiennych wizualizacyjnych*)
rtbDispencer34EnableShow		(CLK:=VIS.bDispencer3EnableShow OR VIS.bDispencer4EnableShow,Q=>);
IF rtbDispencer34EnableShow.Q THEN	
	VIS.bDispencer3EnableShow 	:= TRUE;	
	VIS.bDispencer4EnableShow 	:= TRUE;		
END_IF
ftbDispencer34EnableShow		(CLK:=VIS.bDispencer3EnableShow  AND VIS.bDispencer4EnableShow,Q=>);
IF ftbDispencer34EnableShow.Q THEN	
	VIS.bDispencer3EnableShow 	:= FALSE;	
	VIS.bDispencer4EnableShow 	:= FALSE;	
END_IF
END_ACTION

ACTION aDispencersLiftersAfter:
eDispencer1State;
eDispencer2State;
eDispencer3State;
eDispencer4State;
VIS.lrDispencersCatchHeightCV;

// TACKA OKAPOWA // wysterowana gdy któryś z bloków dozowników włączy
QbDispencer1DropCatcherValveActuator	:=	(bDispencer1DropCatcherValveActuator AND bDispencer2DropCatcherValveActuator) AND NOT (fbDispencersCatch1Station.eState = E_Station.eHoming);
QbDispencer2DropCatcherValveActuator	:=	(bDispencer2DropCatcherValveActuator AND bDispencer1DropCatcherValveActuator) AND NOT (fbDispencersCatch1Station.eState = E_Station.eHoming);
QbDispencer3DropCatcherValveActuator	:=	(bDispencer3DropCatcherValveActuator AND bDispencer4DropCatcherValveActuator) AND NOT (fbDispencersCatch1Station.eState = E_Station.eHoming);
QbDispencer4DropCatcherValveActuator	:=	(bDispencer4DropCatcherValveActuator AND bDispencer3DropCatcherValveActuator) AND NOT (fbDispencersCatch1Station.eState = E_Station.eHoming);

IF VIS.bDispencer1Dose AND NOT bDispencer1DropCatcherValveActuator THEN
	QbDispencer2DropCatcherValveActuator := FALSE;
END_IF
IF VIS.bDispencer2Dose AND NOT bDispencer2DropCatcherValveActuator THEN
	QbDispencer1DropCatcherValveActuator := FALSE;
END_IF
IF VIS.bDispencer3Dose AND NOT bDispencer3DropCatcherValveActuator THEN
	QbDispencer4DropCatcherValveActuator := FALSE;
END_IF
IF VIS.bDispencer4Dose AND NOT bDispencer4DropCatcherValveActuator THEN
	QbDispencer3DropCatcherValveActuator := FALSE;
END_IF

(*Przekazywnaie sygnałów osi na rzeczywistą*)
// DOZOWNIKI 1-2
IF  bDispenser1LifterMaster THEN
	aDispencerLifter12AxisRef := aDispenser1VirtualLifter;
ELSIF bDispenser2LifterMaster THEN
	aDispencerLifter12AxisRef := aDispenser2VirtualLifter;
END_IF

// DOZOWNIKI 3-4
IF  bDispenser3LifterMaster THEN
	aDispencerLifter34AxisRef := aDispenser3VirtualLifter;
ELSIF bDispenser4LifterMaster THEN
	aDispencerLifter34AxisRef := aDispenser4VirtualLifter;
END_IF
END_ACTION

ACTION aDispencersLiftersBefore:

(*Zmienne które synchornizują rozpoczęcie dozowania, czyli jak podnośnik jest na dole*)
(*w tym momencie ma zacząć się 1 faza dozowania, wystawiane w ePreparingToDose*)
(*bDispenser1MultiMasterSyncOut jest wystawiany w ePreparingToDose od skończonego ruchu zasysania oraz pozycji podnośnika*)
bDispencer12MultiMasterSync	:=		(NOT bDispencer1Enable OR bDispenser1MultiMasterSyncOut OR NOT VIS.bDispencer1Dose) AND 
									(NOT bDispencer2Enable OR bDispenser2MultiMasterSyncOut OR NOT VIS.bDispencer2Dose) ;

bDispencer34MultiMasterSync	:=		(NOT bDispencer3Enable OR bDispenser3MultiMasterSyncOut OR NOT VIS.bDispencer3Dose)  AND
									(NOT bDispencer4Enable OR bDispenser4MultiMasterSyncOut OR NOT VIS.bDispencer4Dose) ;
P02_DispencersCharts.bDispencersSyncSim	:=NOT P02_DispencersCharts.fbDisp.bEnable OR NOT P02_DispencersCharts.bDispenserSimMultiMasterSyncOut OR NOT P02_DispencersCharts.fbDisp.bRun;																 									 
// DOZOWNIKI 1-2
(*Przypisanie rzeczywistych osi do akualnych*)
aDispenser1VirtualLifter	:=	aDispencerLifter12AxisRef;
aDispenser2VirtualLifter	:=	aDispencerLifter12AxisRef;

(*Zsumowanie przycisków od przeciągnia, do skrócenia IFów*)
bDispencer1Manual:=VIS.bDispencer12ManualLifterUp OR VIS.bDispencer12ManualLifterDown OR VIS.bDispencer1PullingFast OR VIS.bDispencer1PullingSlow OR VIS.bDispencer1Dose;
bDispencer2Manual:=VIS.bDispencer12ManualLifterUp OR VIS.bDispencer12ManualLifterDown OR VIS.bDispencer2PullingFast OR VIS.bDispencer2PullingSlow OR VIS.bDispencer2Dose;

(*BEFORE*)
(*Przekazywanie kontroli przez odpowiedni blok zależnie od stanów*)
(*Priorytet ma dozownika 1*)
IF  eDispencer1State<>E_Station.eDisabled  AND ((eDispencer1State<>E_Station.eReady AND NOT (eDispencer1State=E_Station.eManualMovement))  OR (eDispencer1State=E_Station.eManualMovement AND bDispencer1Manual)) THEN
		bDispencer1WithLifter	:=	TRUE;
		bDispencer2WithLifter	:= FALSE;
		bDispenser1LifterMaster	:= TRUE;
		bDispenser2LifterMaster	:= FALSE;
ELSIF  eDispencer2State<>E_Station.eDisabled  AND (eDispencer2State<>E_Station.eReady AND NOT (eDispencer2State=E_Station.eManualMovement) OR (eDispencer2State=E_Station.eManualMovement AND bDispencer2Manual)) THEN
		bDispencer2WithLifter	:=	TRUE;
		bDispencer1WithLifter	:= FALSE;
		bDispenser2LifterMaster	:= TRUE;
		bDispenser1LifterMaster	:= FALSE;
END_IF

// DOZOWNIKI 3-4
aDispenser3VirtualLifter	:=	aDispencerLifter34AxisRef;
aDispenser4VirtualLifter	:=	aDispencerLifter34AxisRef;

(*Zsumowanie przycisków od przeciągnia, do skrócenia IFów*)
bDispencer3Manual:=VIS.bDispencer34ManualLifterUp OR VIS.bDispencer34ManualLifterDown OR VIS.bDispencer3PullingFast OR VIS.bDispencer3PullingSlow OR VIS.bDispencer3Dose;
bDispencer4Manual:=VIS.bDispencer34ManualLifterUp OR VIS.bDispencer34ManualLifterDown OR VIS.bDispencer4PullingFast OR VIS.bDispencer4PullingSlow OR VIS.bDispencer4Dose;

IF  eDispencer3State<>E_Station.eDisabled  AND ((eDispencer3State<>E_Station.eReady AND NOT (eDispencer3State=E_Station.eManualMovement))  OR (eDispencer3State=E_Station.eManualMovement AND bDispencer3Manual)) THEN
	bDispencer3WithLifter	:=	TRUE;
	bDispencer4WithLifter	:= FALSE;
	bDispenser3LifterMaster	:= TRUE;
	bDispenser4LifterMaster	:= FALSE;
ELSIF  eDispencer4State<>E_Station.eDisabled  AND (eDispencer4State<>E_Station.eReady AND NOT (eDispencer4State=E_Station.eManualMovement) OR (eDispencer4State=E_Station.eManualMovement AND bDispencer4Manual)) THEN
	bDispencer4WithLifter	:=	TRUE;
	bDispencer3WithLifter	:= FALSE;	
	bDispenser4LifterMaster	:= TRUE;
	bDispenser3LifterMaster	:= FALSE;
END_IF
END_ACTION

ACTION aDispencersManualMode:
(*
Nazwa:			aDispencersManualMode
Opis:			
Wersja:			v0.2
Data:			2024-03-11
Autor:			DP
Urzadzenia:		Dozowniki
Konfiguracja:	
Zmiany:
20230311 - [DP] Sycnhronizacja pod nowa wizke
20230303 - Dodany ft Continous
Info:
*)

VIS.bDispencersManualLifterUp;   	
VIS.bDispencersManualLifterDown;
VIS.bDispencersPullingFast;  	
VIS.bDispencersPullingSlow;   	
ftbDispencersPullingSlow(CLK:=VIS.bDispencersPullingSlow, Q=>);
ftbDispencersPullingFast(CLK:=VIS.bDispencersPullingFast, Q=>);
ftbDispencersPullingSlowContinous(CLK:=VIS.bDispencersPullingSlowContinous, Q=>);
ftbDispencersPullingFastContinous(CLK:=VIS.bDispencersPullingFastContinous, Q=>);
ftbDispencersLifterUp(CLK:=VIS.bDispencersManualLifterUp, Q=>);
ftbDispencersLifterDown(CLK:=VIS.bDispencersManualLifterDown, Q=>);

IF ftbDispencersPullingSlow.Q OR ftbDispencersPullingFast.Q THEN
	VIS.bDispencer1PullingFast:=FALSE;
	VIS.bDispencer2PullingFast:=FALSE; 
	VIS.bDispencer3PullingFast:=FALSE; 	
	VIS.bDispencer4PullingFast:=FALSE; 		
	VIS.bDispencer1PullingSlow:=FALSE; 
	VIS.bDispencer2PullingSlow:=FALSE; 
	VIS.bDispencer3PullingSlow:=FALSE; 
	VIS.bDispencer4PullingSlow:=FALSE; 	
	VIS.bDispencersPullingFast:=FALSE;
	VIS.bDispencersPullingSlow:=FALSE;
END_IF

IF ftbDispencersPullingSlowContinous.Q OR ftbDispencersPullingFastContinous.Q THEN
	VIS.bDispencer1PullingFast:=FALSE;
	VIS.bDispencer2PullingFast:=FALSE; 
	VIS.bDispencer3PullingFast:=FALSE; 	
	VIS.bDispencer4PullingFast:=FALSE; 		
	VIS.bDispencer1PullingSlow:=FALSE; 
	VIS.bDispencer2PullingSlow:=FALSE; 
	VIS.bDispencer3PullingSlow:=FALSE; 
	VIS.bDispencer4PullingSlow:=FALSE; 	
	VIS.bDispencersPullingFast:=FALSE;
	VIS.bDispencersPullingSlow:=FALSE;
END_IF


IF ftbDispencersLifterUp.Q OR ftbDispencersLifterDown.Q THEN
	VIS.bDispencer12ManualLifterUp := FALSE;
	VIS.bDispencer34ManualLifterUp := FALSE;
	
	VIS.bDispencer12ManualLifterDown :=  FALSE;
	VIS.bDispencer34ManualLifterDown :=  FALSE;
END_IF

(*VIS.bDispencer12ManualLifterUp := VIS.bDispencer12ManualLifterUp OR VIS.bDispencersManualLifterUp;
VIS.bDispencer34ManualLifterUp := VIS.bDispencer34ManualLifterUp OR VIS.bDispencersManualLifterUp;

VIS.bDispencer12ManualLifterDown := VIS.bDispencer12ManualLifterDown OR VIS.bDispencersManualLifterDown;
VIS.bDispencer34ManualLifterDown := VIS.bDispencer34ManualLifterDown OR VIS.bDispencersManualLifterDown;

(VIS.bDispencer1PullingFast	:= VIS.bDispencer1PullingFast OR VIS.bDispencersPullingFast OR VIS.bDispencersPullingFastContinous;
VIS.bDispencer2PullingFast	:= VIS.bDispencer2PullingFast OR VIS.bDispencersPullingFast OR VIS.bDispencersPullingFastContinous;
VIS.bDispencer3PullingFast	:= VIS.bDispencer3PullingFast OR VIS.bDispencersPullingFast OR VIS.bDispencersPullingFastContinous;
VIS.bDispencer4PullingFast	:= VIS.bDispencer4PullingFast OR VIS.bDispencersPullingFast OR VIS.bDispencersPullingFastContinous;

VIS.bDispencer1PullingSlow	:= VIS.bDispencer1PullingSlow OR VIS.bDispencersPullingSlow OR VIS.bDispencersPullingSlowContinous;
VIS.bDispencer2PullingSlow	:= VIS.bDispencer2PullingSlow OR VIS.bDispencersPullingSlow OR VIS.bDispencersPullingSlowContinous;
VIS.bDispencer3PullingSlow	:= VIS.bDispencer3PullingSlow OR VIS.bDispencersPullingSlow OR VIS.bDispencersPullingSlowContinous;
VIS.bDispencer4PullingSlow	:= VIS.bDispencer4PullingSlow OR VIS.bDispencersPullingSlow OR VIS.bDispencersPullingSlowContinous;
*)

(*Przeciąganie ciągłe przez 30sekund*)
IF VIS.bDispencersPullingFastContinous THEN
	VIS.bDispencersPullingFast	:=	TRUE;
END_IF
IF VIS.bDispencersPullingSlowContinous THEN
	VIS.bDispencersPullingSlow	:=	TRUE;
END_IF

tonbDispencersPullingContinous	(IN:=VIS.bDispencersPullingFastContinous OR VIS.bDispencersPullingSlowContinous, PT:=T#30S);
IF tonbDispencersPullingContinous.Q THEN
	VIS.bDispencersPullingFastContinous	:=	FALSE;	
	VIS.bDispencersPullingSlowContinous	:=	FALSE;	
	VIS.bDispencersPullingFast			:=	FALSE;
	VIS.bDispencersPullingSlow			:=	FALSE;
END_IF


(**************** Synch z UBL************************)
//Domyślnie katywne 3 dozowniki
rtManualMode			(CLK:=P00_PackML.fbPMLModeManager.eModeStatus = Tc3_PackML.E_PMLUnitMode.ePMLUnitMode_MANUAL,Q=>);
ftManualMode			(CLK:=P00_PackML.fbPMLModeManager.eModeStatus = Tc3_PackML.E_PMLUnitMode.ePMLUnitMode_MANUAL,Q=>);
rtbDispencer1Sync		(CLK:=VIS.bDispencer1Sync,Q=>);
rtbDispencer2Sync		(CLK:=VIS.bDispencer2Sync,Q=>);
rtbDispencer3Sync		(CLK:=VIS.bDispencer3Sync,Q=>);
rtbDispencer4Sync		(CLK:=VIS.bDispencer4Sync,Q=>);
rtbDispencer12Sync		(CLK:=VIS.bDispencer12Sync,Q=>);
rtbDispencer34Sync		(CLK:=VIS.bDispencer34Sync,Q=>);
rtbDispencer1234Sync	(CLK:=VIS.bDispencer1234Sync,Q=>);


IF rtbDispencer1Sync.Q THEN			
	VIS.bDispencer1Sync		:=	TRUE;
	VIS.bDispencer2Sync		:=	FALSE;
	VIS.bDispencer3Sync		:=	FALSE;	
	VIS.bDispencer4Sync		:=	FALSE;	
	VIS.bDispencer12Sync	:=	FALSE;
	VIS.bDispencer34Sync	:=	FALSE;
	VIS.bDispencer1234Sync	:=	FALSE;
		bDispencer1SyncTemp	:=	TRUE;
		bDispencer2SyncTemp	:=	FALSE;
		bDispencer3SyncTemp	:=	FALSE;
		bDispencer4SyncTemp	:=	FALSE;	
END_IF
IF rtbDispencer2Sync.Q THEN			
	VIS.bDispencer1Sync		:=	FALSE;
	VIS.bDispencer2Sync		:=	TRUE;
	VIS.bDispencer3Sync		:=	FALSE;	
	VIS.bDispencer4Sync		:=	FALSE;	
	VIS.bDispencer12Sync	:=	FALSE;
	VIS.bDispencer34Sync	:=	FALSE;
	VIS.bDispencer1234Sync	:=	FALSE;
		bDispencer1SyncTemp	:=	FALSE;
		bDispencer2SyncTemp	:=	TRUE;
		bDispencer3SyncTemp	:=	FALSE;
		bDispencer4SyncTemp	:=	FALSE;	
END_IF
IF rtbDispencer3Sync.Q THEN			
	VIS.bDispencer1Sync		:=	FALSE;
	VIS.bDispencer2Sync		:=	FALSE;
	VIS.bDispencer3Sync		:=	TRUE;
	VIS.bDispencer4Sync		:=	FALSE;	
	VIS.bDispencer12Sync	:=	FALSE;
	VIS.bDispencer34Sync	:=	FALSE;
	VIS.bDispencer1234Sync	:=	FALSE;
		bDispencer1SyncTemp	:=	FALSE;
		bDispencer2SyncTemp	:=	FALSE;
		bDispencer3SyncTemp	:=	TRUE;
		bDispencer4SyncTemp	:=	FALSE;	
END_IF
IF rtbDispencer4Sync.Q THEN			
	VIS.bDispencer1Sync		:=	FALSE;
	VIS.bDispencer2Sync		:=	FALSE;
	VIS.bDispencer3Sync		:=	FALSE;
	VIS.bDispencer4Sync		:=	TRUE;
	VIS.bDispencer12Sync	:=	FALSE;
	VIS.bDispencer34Sync	:=	FALSE;
	VIS.bDispencer1234Sync	:=	FALSE;
		bDispencer1SyncTemp	:=	FALSE;
		bDispencer2SyncTemp	:=	FALSE;
		bDispencer3SyncTemp	:=	FALSE;
		bDispencer4SyncTemp	:=	TRUE;	
END_IF
IF rtbDispencer12Sync.Q THEN			
	VIS.bDispencer1Sync		:=	FALSE;
	VIS.bDispencer2Sync		:=	FALSE;
	VIS.bDispencer3Sync		:=	FALSE;
	VIS.bDispencer4Sync		:=	FALSE;
	VIS.bDispencer12Sync	:=	TRUE;
	VIS.bDispencer34Sync	:=	FALSE;
	VIS.bDispencer1234Sync	:=	FALSE;
		bDispencer1SyncTemp	:=	TRUE;
		bDispencer2SyncTemp	:=	TRUE;
		bDispencer3SyncTemp	:=	FALSE;
		bDispencer4SyncTemp	:=	FALSE;	
END_IF
IF rtbDispencer34Sync.Q THEN			
	VIS.bDispencer1Sync		:=	FALSE;
	VIS.bDispencer2Sync		:=	FALSE;
	VIS.bDispencer3Sync		:=	FALSE;
	VIS.bDispencer4Sync		:=	FALSE;
	VIS.bDispencer12Sync	:=	FALSE;
	VIS.bDispencer34Sync	:=	TRUE;
	VIS.bDispencer1234Sync	:=	FALSE;
		bDispencer1SyncTemp	:=	FALSE;
		bDispencer2SyncTemp	:=	FALSE;
		bDispencer3SyncTemp	:=	TRUE;
		bDispencer4SyncTemp	:=	TRUE;		
END_IF
IF rtbDispencer1234Sync.Q THEN			
	VIS.bDispencer1Sync		:=	FALSE;
	VIS.bDispencer2Sync		:=	FALSE;
	VIS.bDispencer3Sync		:=	FALSE;
	VIS.bDispencer4Sync		:=	FALSE;
	VIS.bDispencer12Sync	:=	FALSE;
	VIS.bDispencer34Sync	:=	FALSE;
	VIS.bDispencer1234Sync	:=	TRUE;
		bDispencer1SyncTemp	:=	TRUE;
		bDispencer2SyncTemp	:=	TRUE;
		bDispencer3SyncTemp	:=	TRUE;
		bDispencer4SyncTemp	:=	TRUE;		
END_IF
IF rtManualMode.Q THEN				
	VIS.bDispencer1Sync		:=	FALSE;
	VIS.bDispencer2Sync		:=	FALSE;
	VIS.bDispencer3Sync		:=	FALSE;	
	VIS.bDispencer4Sync		:=	FALSE;	
	VIS.bDispencer12Sync	:=	FALSE;
	VIS.bDispencer34Sync	:=	FALSE;
	VIS.bDispencer1234Sync	:=	TRUE;
	//	bDispencer1SyncTemp	:=	TRUE;
	//	bDispencer2SyncTemp	:=	TRUE;
	//	bDispencer3SyncTemp	:=	TRUE;
	//	bDispencer4SyncTemp	:=	TRUE;		
END_IF
IF ftManualMode.Q THEN
	VIS.bDispencer1234Sync	:=	FALSE;
	VIS.bDispencer1Sync		:=	FALSE;	
	VIS.bDispencer2Sync		:=	FALSE;	
	VIS.bDispencer3Sync		:=	FALSE;
	VIS.bDispencer4Sync		:=	FALSE;
	VIS.bDispencer12Sync	:=	FALSE;
	VIS.bDispencer34Sync	:=	FALSE;
	VIS.bDispencer1234Sync	:=	FALSE;
		bDispencer1SyncTemp	:=	FALSE;
		bDispencer2SyncTemp	:=	FALSE;
		bDispencer3SyncTemp	:=	FALSE;
		bDispencer4SyncTemp	:=	FALSE;
END_IF

fbDispencer1Sync(bIn:=bDispencer1SyncTemp, tFilterTimeon:=T#1S, tFilterTimeOff:=T#1S);
fbDispencer2Sync(bIn:=bDispencer2SyncTemp, tFilterTimeon:=T#1S, tFilterTimeOff:=T#1S);
fbDispencer3Sync(bIn:=bDispencer3SyncTemp, tFilterTimeon:=T#1S, tFilterTimeOff:=T#1S);
fbDispencer4Sync(bIn:=bDispencer4SyncTemp, tFilterTimeon:=T#1S, tFilterTimeOff:=T#1S);

//Trigery po zmianie dozownika
rtDispencer1Sync	(CLK:=fbDispencer1Sync.bOut,Q=>);
rtDispencer2Sync	(CLK:=fbDispencer2Sync.bOut,Q=>);
rtDispencer3Sync	(CLK:=fbDispencer3Sync.bOut,Q=>);
rtDispencer4Sync	(CLK:=fbDispencer4Sync.bOut,Q=>);

rtHeightSetDispencer12(CLK:=VIS.bDispencersHeightSet AND (fbDispencer1Sync.bOUT OR fbDispencer2Sync.bOut)	, Q=>);
rtHeightSetDispencer34(CLK:=VIS.bDispencersHeightSet AND (fbDispencer3Sync.bOut OR fbDispencer4Sync.bOut)	, Q=>);


//Opóźnienie po zmianie, zabezpieczenie przed zbyt szybką zmianą 
tofDispencersSync	(IN:=rtDispencer1Sync.Q OR rtDispencer2Sync.Q OR rtDispencer3Sync.Q OR rtDispencer4Sync.Q,	PT:=T#1S);

